Yaskawa INFORM job: X2_38-47,64(2)(90,0).JBI

/JOB
//NAME X2_38-47,64(2)(90,0)
//POS
///NPOS 774,774,774,27,0,0
///TOOL 0
///POSTYPE PULSE
///PULSE
C00000=-10776,-116726,-133110,1428,79202,268
C00001=-117551,-99167,-129064,14869,107235,27560
C00002=-118060,-97833,-124544,14759,105287,27149
C00003=-118255,-97731,-122391,14687,104086,26936
C00004=-118255,-99005,-121658,14606,103015,26804
C00005=-118252,-98719,-121832,14623,103261,26835
C00006=-118753,-92238,-119382,14829,105109,26899
C00007=-118252,-98719,-121832,14623,103261,26835
C00008=-117548,-101379,-128390,14732,105732,27372
C00009=-119930,-99721,-129265,15188,107465,26816
C00010=-120369,-98285,-124713,15062,105542,26424
C00011=-120537,-98252,-122491,14975,104264,26206
C00012=-120537,-99415,-121812,14899,103281,26083
C00013=-120552,-99088,-121997,14922,103557,26112
C00014=-120983,-92542,-119530,15124,105413,26206
C00015=-120552,-99088,-121997,14922,103557,26112
C00016=-119945,-101871,-128593,15052,105999,26622
C00017=-126449,-117484,-130445,19479,74849,30062
C00018=-126433,-122162,-123583,20167,68593,29001
C00019=-126700,-111661,-117040,20113,69946,29141
C00020=-126798,-108107,-114012,20160,69935,29102
C00021=-126799,-108400,-113008,20254,69212,28975
C00022=-126718,-108336,-113627,20168,69582,29070
C00023=-124486,-105728,-112699,19107,69790,29924
C00024=-126718,-108336,-113627,20168,69582,29070
C00025=-121607,-132044,-121280,18982,61321,29585
C00026=-106120,-105771,-112642,10491,66484,36125
C00027=-107709,-101450,-111061,11179,67916,35692
C00028=-106120,-105771,-112642,10491,66484,36125
C00029=-113778,-131562,-126460,14735,63009,32904
C00030=-125989,-135705,-128836,15868,81833,-19678
C00031=-122637,-125595,-122855,15098,82666,-18409
C00032=-121382,-121958,-120533,14807,82865,-17952
C00033=-121382,-122071,-118910,14836,81841,-18076
C00034=-121382,-121958,-120533,14807,82865,-17952
C00035=-106979,-143901,-125029,2861,68009,-11090
C00036=-108002,-136905,-123073,3147,70435,-11396
C00037=-106979,-143901,-125029,2861,68009,-11090
C00038=-130918,-93362,-108301,23503,98063,-21430
C00039=-128613,-93045,-108174,23197,97523,-20724
C00040=-130918,-93362,-108301,23503,98063,-21430
C00041=-136165,-97259,-113946,24281,100844,-22722
C00042=-136175,-89641,-119549,25205,107565,-21267
C00043=-114744,-130738,-127344,-18726,86415,24127
C00044=-118651,-123075,-122041,-18017,86194,22796
C00045=-120132,-120263,-119410,-17742,85711,22351
C00046=-120132,-120365,-118339,-17753,85031,22450
C00047=-120131,-120316,-118616,-17749,85218,22423
C00048=-120610,-114014,-116540,-17635,86988,22001
C00049=-120131,-120316,-118616,-17749,85218,22423
C00050=-120535,-116966,-117470,-17658,86102,22155
C00051=-123144,-118008,-117813,-17156,85246,21372
C00052=-120535,-116966,-117470,-17658,86102,22155
C00053=-115268,-126863,-124750,-18631,86672,23904
C00054=-115290,-123417,-132013,-18678,92595,22992
C00055=-123593,-125758,-130163,6995,115060,-67946
C00056=-111289,-112434,-124190,9231,117016,-63234
C00057=-105837,-112853,-120878,9823,114178,-61462
C00058=-105837,-113368,-119803,9744,113264,-61541
C00059=-105837,-112984,-120626,9804,113958,-61481
C00060=-104314,-115180,-121361,9954,113110,-60999
C00061=-105837,-112984,-120626,9804,113958,-61481
C00062=-140180,-156270,-135194,3647,103600,-74458
C00063=-143876,-158808,-133483,2421,103143,-75779
C00064=-143876,-157752,-132173,2418,102880,-75785
C00065=-143876,-158999,-133717,2421,103190,-75779
C00066=-142833,-166242,-135523,2599,100548,-75469
C00067=-143876,-158999,-133717,2421,103190,-75779
C00068=-138517,-137739,-134524,3768,114393,-73549
C00069=-143641,-117492,-131018,10110,103710,-40081
C00070=-127017,-112123,-129453,9078,98380,-24722
C00071=-128303,-122732,-125182,9622,82824,-11347
C00072=-126354,-112603,-118881,9097,83916,-10616
C00073=-125631,-108986,-116438,8904,84188,-10357
C00074=-125631,-109537,-114964,8919,83013,-10441
C00075=-125631,-108986,-116438,8904,84188,-10357
C00076=-110037,-120252,-118594,-5441,76700,-4050
C00077=-111650,-115152,-116920,-4919,78183,-4659
C00078=-110037,-120252,-118594,-5441,76700,-4050
C00079=-125797,-107165,-114352,8951,83863,-10435
C00080=-123589,-104463,-113383,8361,84418,-9668
C00081=-125797,-107165,-114352,8951,83863,-10435
C00082=-128447,-120300,-122969,9661,82730,-11402
C00083=-128462,-115265,-129707,9620,89375,-10895
C00084=-116938,-126430,-125851,-12631,81878,14685
C00085=-119474,-116309,-119688,-11957,82879,13726
C00086=-120416,-112800,-116898,-11714,82830,13413
C00087=-120416,-113088,-115771,-11732,82005,13491
C00088=-121130,-109897,-115487,-11517,83341,13125
C00089=-121652,-107697,-114715,-11371,83913,12898
C00090=-120385,-110630,-116263,-11708,83544,13356
C00091=-116898,-126708,-125088,-12658,81285,14759
C00092=-116961,-121523,-133241,-12544,88781,13978
C00093=-110477,-156196,-127656,-40514,54336,55405
C00094=-116757,-147091,-123275,-37008,53079,52657
C00095=-119129,-143495,-121504,-35581,52690,51595
C00096=-122199,-143523,-121511,-34086,51426,50520
C00097=-119129,-143495,-121504,-35581,52690,51595
C00098=-121389,-143526,-121523,-34489,51757,50806
C00099=-121378,-138155,-118828,-34021,52680,50458
C00100=-121389,-143526,-121523,-34489,51757,50806
C00101=-121337,-120057,-120260,-30579,61379,47564
C00102=-120272,-114318,-116759,-30898,62447,47698
C00103=-120254,-119054,-117181,-31500,60580,48280
C00104=-120272,-114318,-116759,-30898,62447,47698
C00105=-110477,-159292,-131347,-40206,54861,55162
C00106=-115322,-144881,-127675,-10917,26238,44128
C00107=-131784,-127965,-127002,28991,89678,26741
C00108=-120831,-123140,-121731,27130,85392,29797
C00109=-120549,-120601,-118843,27089,84879,29783
C00110=-120549,-120670,-117777,27109,84260,29640
C00111=-120517,-120686,-117908,27101,84315,29665
C00112=-120983,-114470,-115866,27142,86197,29928
C00113=-120517,-120686,-117908,27101,84315,29665
C00114=-121539,-130455,-126219,27290,84728,29379
C00115=-123491,-138727,-133578,17593,86073,29901
C00116=-123873,-130565,-127363,17655,86508,29830
C00117=-124019,-127789,-124130,17687,86001,29706
C00118=-124019,-127817,-123341,17694,85524,29637
C00119=-124041,-127842,-123499,17696,85609,29642
C00120=-124402,-120732,-121277,17740,87868,29843
C00121=-124041,-127842,-123499,17696,85609,29642
C00122=-123895,-130695,-125894,17671,85585,29689
C00123=-123514,-138829,-132098,17610,85158,29761
C00124=-131669,-108309,-130646,31875,113573,61343
C00125=-139138,-132176,-121475,37127,109735,76690
C00126=-136347,-141301,-121131,36509,104575,76083
C00127=-135137,-144527,-120818,36387,102556,75910
C00128=-135139,-143303,-118803,36292,102059,75739
C00129=-135137,-144527,-120818,36387,102556,75910
C00130=-123222,-117207,-112602,33876,112841,80142
C00131=-123302,-123100,-114500,33386,111310,79603
C00132=-123222,-117207,-112602,33876,112841,80142
C00133=-149473,-167599,-122340,40123,93659,70303
C00134=-145955,-169881,-122827,40768,91382,70949
C00135=-149473,-167599,-122340,40123,93659,70303
C00136=-154660,-158984,-124630,39692,100555,70658
C00137=-145602,-129354,-130944,11561,117970,66438
C00138=-141571,-135796,-129141,-17923,112920,58745
C00139=-145358,-145317,-128855,-18021,107261,58200
C00140=-146973,-148537,-128532,-18134,105137,57926
C00141=-146977,-147425,-126561,-18072,104525,58019
C00142=-146951,-147398,-126788,-18082,104677,58005
C00143=-148016,-155121,-128806,-18044,101844,58047
C00144=-146951,-147398,-126788,-18082,104677,58005
C00145=-147811,-154474,-129578,-18071,102659,57998
C00146=-150760,-151393,-128781,-18698,103033,56852
C00147=-147811,-154474,-129578,-18071,102659,57998
C00148=-142197,-142429,-130522,-17697,110344,58914
C00149=-120703,-123129,-132845,19094,121060,67264
C00150=-120658,-146832,-128060,18624,118943,66884
C00151=-120634,-158899,-128202,17585,113113,65913
C00152=-120623,-163194,-128036,17271,110903,65572
C00153=-120623,-161024,-125795,17237,110651,65534
C00154=-120562,-161261,-126266,17282,110799,65580
C00155=-120543,-169070,-128088,16945,108025,65171
C00156=-120562,-161261,-126266,17282,110799,65580
C00157=-120603,-145779,-126506,18564,118536,66834
C00158=-125859,-133715,-124767,32608,106843,81797
C00159=-122845,-142953,-124347,32149,101432,81430
C00160=-121547,-146160,-123992,32074,99345,81353
C00161=-121546,-144979,-121994,32008,98813,81200
C00162=-109812,-115651,-114700,28773,111647,86169
C00163=-109420,-121743,-116686,28433,109829,85843
C00164=-109812,-115651,-114700,28773,111647,86169
C00165=-136113,-171916,-125823,37236,88758,74782
C00166=-132431,-173177,-126093,37775,86796,75630
C00167=-136113,-171916,-125823,37236,88758,74782
C00168=-141699,-164023,-128432,36630,95711,74814
C00169=-125872,-133752,-131219,33440,110189,40846
C00170=-133109,-126295,-132836,15576,121717,-49477
C00171=-134095,-144484,-127159,11413,120192,-39245
C00172=-134095,-142728,-123587,11251,118920,-39381
C00173=-134108,-141028,-121891,11256,119008,-39376
C00174=-115660,-122947,-115610,-13186,126131,-57848
C00175=-119844,-134491,-118750,-17115,121000,-60623
C00176=-133528,-137451,-116046,-34139,108998,-80448
C00177=-134077,-138654,-116284,-35996,107959,-82962
C00178=-134074,-140235,-119255,-36225,108790,-83252
C00179=-128746,-104991,-133081,-28169,117444,-49732
C00180=-123335,-90933,-122081,-14660,102496,-9308
C00181=-120623,-92535,-112214,-7385,88125,11837
C00182=-120622,-94347,-109953,-7392,85821,11972
C00183=-121706,-96320,-109727,-7087,84579,11689
C00184=-119347,-92925,-108176,-7759,85570,12397
C00185=-120623,-94767,-108750,-7400,84873,12029
C00186=-120184,-98406,-104184,11463,70199,-7234
C00187=-120621,-97250,-102226,16251,67423,-11647
C00188=-120622,-96877,-104163,16104,68755,-11460
C00189=-120643,-108357,-118989,16415,66098,-11840
C00190=-67024,-106779,-124945,-13769,92672,20129
C00191=-67015,-109280,-122780,-13735,90127,20415
C00192=-68524,-114997,-123393,-13374,87393,20218
C00193=-67240,-109374,-121326,-13663,89172,20449
C00194=-67101,-109000,-122679,-13716,90193,20379
C00195=-67110,-106486,-124839,-13750,92741,20094
C00196=-120616,-103713,-129855,-8435,78518,79847
C00197=-120615,-108904,-127553,-8566,74477,80127
C00198=-120827,-110646,-126375,-8530,72852,80171
C00199=-120813,-110572,-126430,-8535,72927,80169
C00200=-120709,-110247,-126307,-8582,73030,80199
C00201=-120779,-110557,-126444,-8550,72945,80181
C00202=-120615,-108909,-127550,-8566,74473,80128
C00203=-118661,-125998,-116417,-35444,53464,49551
C00204=-120918,-122974,-114552,-34038,52889,48644
C00205=-120869,-128815,-114683,-35350,50480,49611
C00206=-120575,-146473,-114035,-40240,44023,53993
C00207=-120599,-119966,-113452,-30276,65744,57931
C00208=-118319,-121507,-115012,-31110,66714,58605
C00209=-113281,-124998,-118777,-32819,69049,60013
C00210=-113467,-117261,-128448,-33027,70743,59318
C00211=-117537,-116112,-134646,-12805,84442,25722
C00212=-120610,-126431,-125414,1040,80197,3464
C00213=-120610,-126707,-122448,1046,78230,3447
C00214=-122238,-127010,-121321,1494,77406,2886
C00215=-120610,-126687,-121221,1049,77486,3441
C00216=-120610,-126294,-121087,1045,77585,3442
C00217=-120610,-126285,-120333,4549,75913,-5215
C00218=-120610,-126340,-121533,4537,76621,-5189
C00219=-125895,-134934,-128716,6057,76967,-6982
C00220=-120648,-124280,-131590,4464,45149,-4941
C00221=-120660,-101129,-132257,5341,102721,-45112
C00222=-120607,-133883,-126281,5735,119700,-79532
C00223=-120606,-133398,-123219,5634,118073,-79618
C00224=-121084,-133632,-122119,5424,117305,-79842
C00225=-121025,-133506,-122086,5447,117346,-79817
C00226=-120605,-133184,-121944,5595,117401,-79652
C00227=-120606,-133121,-120429,13889,116737,-67437
C00228=-120606,-132780,-121444,14001,117514,-67337
C00229=-120606,-133413,-124386,14219,118956,-67146
C00230=-118302,-128282,-130929,25956,92288,-30440
C00231=-120609,-125694,-119256,16594,71477,-14811
C00232=-120609,-125321,-116628,16727,70109,-15005
C00233=-120267,-125069,-115718,16650,69625,-14949
C00234=-120609,-125952,-120025,-8845,76809,6022
C00235=-120609,-125682,-119997,-8842,76927,6012
C00236=-120946,-125172,-117915,-18180,76717,18969
C00237=-120609,-125456,-118894,-18238,77226,19012
C00238=-120610,-125544,-121647,-18141,78796,18775
C00239=-120644,-111765,-129409,-18832,94472,5338
C00240=-120647,-108820,-131188,-26213,120818,-60808
C00241=-120603,-141811,-125437,-24145,112419,-84195
C00242=-120603,-140407,-122244,-23914,111279,-83943
C00243=-120716,-139436,-120851,-23880,110920,-83910
C00244=-120603,-141515,-124307,-1,115345,-75490
C00245=-120603,-141196,-124279,-1,115492,-75490
C00246=-120750,-138616,-117883,30210,107343,-65244
C00247=-120602,-139074,-119094,30337,107734,-65073
C00248=-120603,-140473,-121905,30531,108612,-64825
C00249=-123038,-137969,-128708,31970,112888,-64779
C00250=-147472,-118060,-121113,40576,103304,-81843
C00251=-147472,-118630,-118217,40218,101703,-82475
C00252=-147472,-118727,-117017,40094,101093,-82713
C00253=-147408,-115266,-125424,616,120610,-87255
C00254=-147440,-115512,-125518,608,120541,-87267
C00255=-147454,-115617,-125558,7144,119076,-75809
C00256=-147463,-115686,-125590,12209,115534,-64774
C00257=-147467,-115708,-125608,15036,110623,-54333
C00258=-147465,-115687,-125611,15580,106535,-46817
C00259=-147461,-115654,-125607,15271,104034,-42312
C00260=-147458,-115622,-125603,14500,101619,-37854
C00261=-147455,-115603,-125598,14501,101625,-37852
C00262=-147455,-114670,-126645,14574,102714,-37720
C00263=-147454,-112308,-128585,14752,105047,-37432
C00264=-120607,-127649,-132770,-5702,79300,5510
C00265=-120610,-123519,-126906,-5727,77820,5577
C00266=-120610,-124347,-124400,-5769,75861,5668
C00267=-121328,-123636,-123053,-5535,75349,5445
C00268=-120611,-123827,-123148,-12249,77590,12361
C00269=-120610,-124176,-124804,-8835,80309,9900
C00270=-120610,-124421,-124355,885,77124,6939
C00271=-120609,-123606,-124090,-1533,77411,9469
C00272=-116475,-118028,-122311,-2829,79291,10818
C00273=-112174,-113451,-120859,-4161,80928,12195
C00274=-109550,-110906,-119998,-4966,81848,13023
C00275=-120610,-123835,-125318,-1528,78049,9462
C00276=-120610,-122990,-127374,-1521,79748,9441
C00277=2000,-133752,-131219,0,47993,0
C00278=-10776,-116726,-133110,1428,79202,268
C00279=-117551,-99167,-129064,14869,107235,27560
C00280=-118060,-97833,-124544,14759,105287,27149
C00281=-118255,-97731,-122391,14687,104086,26936
C00282=-118255,-99005,-121658,14606,103015,26804
C00283=-118252,-98719,-121832,14623,103261,26835
C00284=-118753,-92238,-119382,14829,105109,26899
C00285=-118252,-98719,-121832,14623,103261,26835
C00286=-117548,-101379,-128390,14732,105732,27372
C00287=-119930,-99721,-129265,15188,107465,26816
C00288=-120369,-98285,-124713,15062,105542,26424
C00289=-120537,-98252,-122491,14975,104264,26206
C00290=-120537,-99415,-121812,14899,103281,26083
C00291=-120552,-99088,-121997,14922,103557,26112
C00292=-120983,-92542,-119530,15124,105413,26206
C00293=-120552,-99088,-121997,14922,103557,26112
C00294=-119945,-101871,-128593,15052,105999,26622
C00295=-126449,-117484,-130445,19479,74849,30062
C00296=-126433,-122162,-123583,20167,68593,29001
C00297=-126700,-111661,-117040,20113,69946,29141
C00298=-126798,-108107,-114012,20160,69935,29102
C00299=-126799,-108400,-113008,20254,69212,28975
C00300=-126718,-108336,-113627,20168,69582,29070
C00301=-124486,-105728,-112699,19107,69790,29924
C00302=-126718,-108336,-113627,20168,69582,29070
C00303=-121607,-132044,-121280,18982,61321,29585
C00304=-106120,-105771,-112642,10491,66484,36125
C00305=-107709,-101450,-111061,11179,67916,35692
C00306=-106120,-105771,-112642,10491,66484,36125
C00307=-113778,-131562,-126460,14735,63009,32904
C00308=-125989,-135705,-128836,15868,81833,-19678
C00309=-122637,-125595,-122855,15098,82666,-18409
C00310=-121382,-121958,-120533,14807,82865,-17952
C00311=-121382,-122071,-118910,14836,81841,-18076
C00312=-121382,-121958,-120533,14807,82865,-17952
C00313=-106979,-143901,-125029,2861,68009,-11090
C00314=-108002,-136905,-123073,3147,70435,-11396
C00315=-106979,-143901,-125029,2861,68009,-11090
C00316=-130918,-93362,-108301,23503,98063,-21430
C00317=-128613,-93045,-108174,23197,97523,-20724
C00318=-130918,-93362,-108301,23503,98063,-21430
C00319=-136165,-97259,-113946,24281,100844,-22722
C00320=-136175,-89641,-119549,25205,107565,-21267
C00321=-114744,-130738,-127344,-18726,86415,24127
C00322=-118651,-123075,-122041,-18017,86194,22796
C00323=-120132,-120263,-119410,-17742,85711,22351
C00324=-120132,-120365,-118339,-17753,85031,22450
C00325=-120131,-120316,-118616,-17749,85218,22423
C00326=-120610,-114014,-116540,-17635,86988,22001
C00327=-120131,-120316,-118616,-17749,85218,22423
C00328=-120535,-116966,-117470,-17658,86102,22155
C00329=-123144,-118008,-117813,-17156,85246,21372
C00330=-120535,-116966,-117470,-17658,86102,22155
C00331=-115268,-126863,-124750,-18631,86672,23904
C00332=-115290,-123417,-132013,-18678,92595,22992
C00333=-123593,-125758,-130163,6995,115060,-67946
C00334=-111289,-112434,-124190,9231,117016,-63234
C00335=-105837,-112853,-120878,9823,114178,-61462
C00336=-105837,-113368,-119803,9744,113264,-61541
C00337=-105837,-112984,-120626,9804,113958,-61481
C00338=-104314,-115180,-121361,9954,113110,-60999
C00339=-105837,-112984,-120626,9804,113958,-61481
C00340=-140180,-156270,-135194,3647,103600,-74458
C00341=-143876,-158808,-133483,2421,103143,-75779
C00342=-143876,-157752,-132173,2418,102880,-75785
C00343=-143876,-158999,-133717,2421,103190,-75779
C00344=-142833,-166242,-135523,2599,100548,-75469
C00345=-143876,-158999,-133717,2421,103190,-75779
C00346=-138517,-137739,-134524,3768,114393,-73549
C00347=-143641,-117492,-131018,10110,103710,-40081
C00348=-127017,-112123,-129453,9078,98380,-24722
C00349=-128303,-122732,-125182,9622,82824,-11347
C00350=-126354,-112603,-118881,9097,83916,-10616
C00351=-125631,-108986,-116438,8904,84188,-10357
C00352=-125631,-109537,-114964,8919,83013,-10441
C00353=-125631,-108986,-116438,8904,84188,-10357
C00354=-110037,-120252,-118594,-5441,76700,-4050
C00355=-111650,-115152,-116920,-4919,78183,-4659
C00356=-110037,-120252,-118594,-5441,76700,-4050
C00357=-125797,-107165,-114352,8951,83863,-10435
C00358=-123589,-104463,-113383,8361,84418,-9668
C00359=-125797,-107165,-114352,8951,83863,-10435
C00360=-128447,-120300,-122969,9661,82730,-11402
C00361=-128462,-115265,-129707,9620,89375,-10895
C00362=-116938,-126430,-125851,-12631,81878,14685
C00363=-119474,-116309,-119688,-11957,82879,13726
C00364=-120416,-112800,-116898,-11714,82830,13413
C00365=-120416,-113088,-115771,-11732,82005,13491
C00366=-121130,-109897,-115487,-11517,83341,13125
C00367=-121652,-107697,-114715,-11371,83913,12898
C00368=-120385,-110630,-116263,-11708,83544,13356
C00369=-116898,-126708,-125088,-12658,81285,14759
C00370=-116961,-121523,-133241,-12544,88781,13978
C00371=-110477,-156196,-127656,-40514,54336,55405
C00372=-116757,-147091,-123275,-37008,53079,52657
C00373=-119129,-143495,-121504,-35581,52690,51595
C00374=-122199,-143523,-121511,-34086,51426,50520
C00375=-119129,-143495,-121504,-35581,52690,51595
C00376=-121389,-143526,-121523,-34489,51757,50806
C00377=-121378,-138155,-118828,-34021,52680,50458
C00378=-121389,-143526,-121523,-34489,51757,50806
C00379=-121337,-120057,-120260,-30579,61379,47564
C00380=-120272,-114318,-116759,-30898,62447,47698
C00381=-120254,-119054,-117181,-31500,60580,48280
C00382=-120272,-114318,-116759,-30898,62447,47698
C00383=-110477,-159292,-131347,-40206,54861,55162
C00384=-115322,-144881,-127675,-10917,26238,44128
C00385=-131784,-127965,-127002,28991,89678,26741
C00386=-120831,-123140,-121731,27130,85392,29797
C00387=-120549,-120601,-118843,27089,84879,29783
C00388=-120549,-120670,-117777,27109,84260,29640
C00389=-120517,-120686,-117908,27101,84315,29665
C00390=-120983,-114470,-115866,27142,86197,29928
C00391=-120517,-120686,-117908,27101,84315,29665
C00392=-121539,-130455,-126219,27290,84728,29379
C00393=-123491,-138727,-133578,17593,86073,29901
C00394=-123873,-130565,-127363,17655,86508,29830
C00395=-124019,-127789,-124130,17687,86001,29706
C00396=-124019,-127817,-123341,17694,85524,29637
C00397=-124041,-127842,-123499,17696,85609,29642
C00398=-124402,-120732,-121277,17740,87868,29843
C00399=-124041,-127842,-123499,17696,85609,29642
C00400=-123895,-130695,-125894,17671,85585,29689
C00401=-123514,-138829,-132098,17610,85158,29761
C00402=-131669,-108309,-130646,31875,113573,61343
C00403=-139138,-132176,-121475,37127,109735,76690
C00404=-136347,-141301,-121131,36509,104575,76083
C00405=-135137,-144527,-120818,36387,102556,75910
C00406=-135139,-143303,-118803,36292,102059,75739
C00407=-135137,-144527,-120818,36387,102556,75910
C00408=-123222,-117207,-112602,33876,112841,80142
C00409=-123302,-123100,-114500,33386,111310,79603
C00410=-123222,-117207,-112602,33876,112841,80142
C00411=-149473,-167599,-122340,40123,93659,70303
C00412=-145955,-169881,-122827,40768,91382,70949
C00413=-149473,-167599,-122340,40123,93659,70303
C00414=-154660,-158984,-124630,39692,100555,70658
C00415=-145602,-129354,-130944,11561,117970,66438
C00416=-141571,-135796,-129141,-17923,112920,58745
C00417=-145358,-145317,-128855,-18021,107261,58200
C00418=-146973,-148537,-128532,-18134,105137,57926
C00419=-146977,-147425,-126561,-18072,104525,58019
C00420=-146951,-147398,-126788,-18082,104677,58005
C00421=-148016,-155121,-128806,-18044,101844,58047
C00422=-146951,-147398,-126788,-18082,104677,58005
C00423=-147811,-154474,-129578,-18071,102659,57998
C00424=-150760,-151393,-128781,-18698,103033,56852
C00425=-147811,-154474,-129578,-18071,102659,57998
C00426=-142197,-142429,-130522,-17697,110344,58914
C00427=-120703,-123129,-132845,19094,121060,67264
C00428=-120658,-146832,-128060,18624,118943,66884
C00429=-120634,-158899,-128202,17585,113113,65913
C00430=-120623,-163194,-128036,17271,110903,65572
C00431=-120623,-161024,-125795,17237,110651,65534
C00432=-120562,-161261,-126266,17282,110799,65580
C00433=-120543,-169070,-128088,16945,108025,65171
C00434=-120562,-161261,-126266,17282,110799,65580
C00435=-120603,-145779,-126506,18564,118536,66834
C00436=-125859,-133715,-124767,32608,106843,81797
C00437=-122845,-142953,-124347,32149,101432,81430
C00438=-121547,-146160,-123992,32074,99345,81353
C00439=-121546,-144979,-121994,32008,98813,81200
C00440=-109812,-115651,-114700,28773,111647,86169
C00441=-109420,-121743,-116686,28433,109829,85843
C00442=-109812,-115651,-114700,28773,111647,86169
C00443=-136113,-171916,-125823,37236,88758,74782
C00444=-132431,-173177,-126093,37775,86796,75630
C00445=-136113,-171916,-125823,37236,88758,74782
C00446=-141699,-164023,-128432,36630,95711,74814
C00447=-125872,-133752,-131219,33440,110189,40846
C00448=-133109,-126295,-132836,15576,121717,-49477
C00449=-134095,-144484,-127159,11413,120192,-39245
C00450=-134095,-142728,-123587,11251,118920,-39381
C00451=-134108,-141028,-121891,11256,119008,-39376
C00452=-115660,-122947,-115610,-13186,126131,-57848
C00453=-119844,-134491,-118750,-17115,121000,-60623
C00454=-133528,-137451,-116046,-34139,108998,-80448
C00455=-134077,-138654,-116284,-35996,107959,-82962
C00456=-134074,-140235,-119255,-36225,108790,-83252
C00457=-128746,-104991,-133081,-28169,117444,-49732
C00458=-123335,-90933,-122081,-14660,102496,-9308
C00459=-120623,-92535,-112214,-7385,88125,11837
C00460=-120622,-94347,-109953,-7392,85821,11972
C00461=-121706,-96320,-109727,-7087,84579,11689
C00462=-119347,-92925,-108176,-7759,85570,12397
C00463=-120623,-94767,-108750,-7400,84873,12029
C00464=-120184,-98406,-104184,11463,70199,-7234
C00465=-120621,-97250,-102226,16251,67423,-11647
C00466=-120622,-96877,-104163,16104,68755,-11460
C00467=-120643,-108357,-118989,16415,66098,-11840
C00468=-67024,-106779,-124945,-13769,92672,20129
C00469=-67015,-109280,-122780,-13735,90127,20415
C00470=-68524,-114997,-123393,-13374,87393,20218
C00471=-67240,-109374,-121326,-13663,89172,20449
C00472=-67101,-109000,-122679,-13716,90193,20379
C00473=-67110,-106486,-124839,-13750,92741,20094
C00474=-120616,-103713,-129855,-8435,78518,79847
C00475=-120615,-108904,-127553,-8566,74477,80127
C00476=-120827,-110646,-126375,-8530,72852,80171
C00477=-120813,-110572,-126430,-8535,72927,80169
C00478=-120709,-110247,-126307,-8582,73030,80199
C00479=-120779,-110557,-126444,-8550,72945,80181
C00480=-120615,-108909,-127550,-8566,74473,80128
C00481=-118661,-125998,-116417,-35444,53464,49551
C00482=-120918,-122974,-114552,-34038,52889,48644
C00483=-120869,-128815,-114683,-35350,50480,49611
C00484=-120575,-146473,-114035,-40240,44023,53993
C00485=-120599,-119966,-113452,-30276,65744,57931
C00486=-118319,-121507,-115012,-31110,66714,58605
C00487=-113281,-124998,-118777,-32819,69049,60013
C00488=-113467,-117261,-128448,-33027,70743,59318
C00489=-117537,-116112,-134646,-12805,84442,25722
C00490=-120610,-126431,-125414,1040,80197,3464
C00491=-120610,-126707,-122448,1046,78230,3447
C00492=-122238,-127010,-121321,1494,77406,2886
C00493=-120610,-126687,-121221,1049,77486,3441
C00494=-120610,-126294,-121087,1045,77585,3442
C00495=-120610,-126285,-120333,4549,75913,-5215
C00496=-120610,-126340,-121533,4537,76621,-5189
C00497=-125895,-134934,-128716,6057,76967,-6982
C00498=-120648,-124280,-131590,4464,45149,-4941
C00499=-120660,-101129,-132257,5341,102721,-45112
C00500=-120607,-133883,-126281,5735,119700,-79532
C00501=-120606,-133398,-123219,5634,118073,-79618
C00502=-121083,-132569,-121808,5443,117663,-79827
C00503=-120607,-132621,-121847,5608,117630,-79641
C00504=-120606,-132785,-121826,5603,117534,-79644
C00505=-120606,-132451,-120233,13920,116954,-67409
C00506=-120606,-132780,-121444,14001,117514,-67337
C00507=-120606,-133413,-124386,14219,118956,-67146
C00508=-118302,-128282,-130929,25956,92288,-30440
C00509=-120609,-125694,-119256,16594,71477,-14811
C00510=-120609,-125321,-116628,16727,70109,-15005
C00511=-120267,-125069,-115718,16650,69625,-14949
C00512=-120609,-125952,-120025,-8845,76809,6022
C00513=-120609,-125682,-119997,-8842,76927,6012
C00514=-120946,-125172,-117915,-18180,76717,18969
C00515=-120609,-125456,-118894,-18238,77226,19012
C00516=-120610,-125544,-121647,-18141,78796,18775
C00517=-120644,-111765,-129409,-18832,94472,5338
C00518=-120647,-108820,-131188,-26213,120818,-60808
C00519=-120603,-141811,-125437,-24145,112419,-84195
C00520=-120603,-140407,-122244,-23914,111279,-83943
C00521=-120716,-139436,-120851,-23880,110920,-83910
C00522=-120603,-141515,-124307,-1,115345,-75490
C00523=-120603,-141196,-124279,-1,115492,-75490
C00524=-120750,-138616,-117883,30210,107343,-65244
C00525=-120602,-139074,-119094,30337,107734,-65073
C00526=-120603,-140473,-121905,30531,108612,-64825
C00527=-123038,-137969,-128708,31970,112888,-64779
C00528=-147472,-118060,-121113,40576,103304,-81843
C00529=-147472,-118630,-118217,40218,101703,-82475
C00530=-147472,-118727,-117017,40094,101093,-82713
C00531=-147408,-115266,-125424,616,120610,-87255
C00532=-147440,-115512,-125518,608,120541,-87267
C00533=-147454,-115617,-125558,7144,119076,-75809
C00534=-147463,-115686,-125590,12209,115534,-64774
C00535=-147467,-115708,-125608,15036,110623,-54333
C00536=-147465,-115687,-125611,15580,106535,-46817
C00537=-147461,-115654,-125607,15271,104034,-42312
C00538=-147458,-115622,-125603,14500,101619,-37854
C00539=-147455,-115603,-125598,14501,101625,-37852
C00540=-147455,-114670,-126645,14574,102714,-37720
C00541=-147454,-112308,-128585,14752,105047,-37432
C00542=-120607,-127649,-132770,-5702,79300,5510
C00543=-120610,-123519,-126906,-5727,77820,5577
C00544=-120610,-124347,-124400,-5769,75861,5668
C00545=-121328,-123636,-123053,-5535,75349,5445
C00546=-120611,-123827,-123148,-12249,77590,12361
C00547=-120610,-124176,-124804,-8835,80309,9900
C00548=-120610,-124421,-124355,885,77124,6939
C00549=-120609,-123606,-124090,-1533,77411,9469
C00550=-116475,-118028,-122311,-2829,79291,10818
C00551=-112174,-113451,-120859,-4161,80928,12195
C00552=-109550,-110906,-119998,-4966,81848,13023
C00553=-120610,-123835,-125318,-1528,78049,9462
C00554=-120610,-122990,-127374,-1521,79748,9441
C00555=2000,-133752,-131219,0,47993,0
C00556=-63459,-114373,-79771,19626,40886,37257
C00557=-120535,67520,37147,4212,69072,67068
C00558=-120830,69446,43417,4422,66227,66858
C00559=-120946,70374,46117,4513,65052,66770
C00560=-120946,70561,47998,4551,63994,66728
C00561=-120946,70374,46117,4513,65052,66770
C00562=-120262,65088,41656,4214,65044,67021
C00563=-120723,68225,45319,4437,64429,66828
C00564=-120262,65088,41656,4214,65044,67021
C00565=-120141,64198,39022,4125,66199,67107
C00566=-119837,62342,32876,3917,69006,67311
C00567=-133022,42545,9302,483,69993,74705
C00568=-133254,43745,14595,601,67354,74612
C00569=-133346,44332,16823,649,66285,74574
C00570=-133347,44228,18372,654,65278,74568
C00571=-133346,44332,16823,649,66285,74574
C00572=-132762,39917,13904,373,65809,74781
C00573=-133123,42775,16905,546,65433,74650
C00574=-132762,39917,13904,373,65809,74781
C00575=-132666,39314,11672,325,66873,74819
C00576=-132425,38068,6360,208,69500,74909
C00577=-155117,5532,-38436,2147,90846,73739
C00578=-181330,90113,53999,1695,94832,75162
C00579=-181479,87228,54387,1703,93114,75089
C00580=-181540,86155,54651,1706,92402,75059
C00581=-181542,86152,56307,1705,91382,75044
C00582=-181540,86155,54651,1706,92402,75059
C00583=-180656,94851,65604,1626,90111,75325
C00584=-181131,94253,66558,1666,89229,75153
C00585=-181349,89885,61022,1686,90394,75096
C00586=-181131,94253,66558,1666,89229,75153
C00587=-181073,95243,66217,1662,89945,75182
C00588=-180930,97948,65680,1651,91663,75253
C00589=-185436,101694,69046,-5553,88631,72150
C00590=-185900,99624,70331,-5496,86754,72076
C00591=-186087,98901,70984,-5475,85971,72047
C00592=-186087,99023,71813,-5476,85523,72066
C00593=-186087,98901,70984,-5475,85971,72047
C00594=-185708,102060,75107,-5528,85087,72214
C00595=-185637,106217,81264,-5546,83447,72310
C00596=-185813,101011,74470,-5516,84934,72189
C00597=-185596,102468,75930,-5543,84801,72264
C00598=-185712,103515,76702,-5528,84853,72223
C00599=-185252,105372,75160,-5578,86780,72294
C00600=-160848,14099,-19058,-268,71131,81958
C00601=-166181,22945,-3449,-1246,81387,-4932
C00602=-165629,27427,7007,-1415,77267,-4702
C00603=-165325,28785,10065,-1509,76088,-4584
C00604=-165325,28859,11250,-1513,75397,-4577
C00605=-165325,28785,10065,-1509,76088,-4584
C00606=-165316,31705,12964,-1515,75805,-4576
C00607=-165325,28785,10065,-1509,76088,-4584
C00608=-158615,35277,16566,-12881,79402,10247
C00609=-158695,35491,17753,-12887,78784,10285
C00610=-159268,36430,18712,-12762,78589,10105
C00611=-158695,35389,16453,-12860,79513,10210
C00612=-158695,35595,7262,-12723,85139,9628
C00613=-159201,23460,163,-1108,64126,82575
C00614=-159224,25290,5934,-1122,61515,82592
C00615=-159868,27923,10103,-801,60293,82359
C00616=-159868,27994,11092,-805,59722,82362
C00617=-159702,23782,6087,-883,60640,82418
C00618=-159324,22038,5481,-1084,60120,82567
C00619=-159393,26328,9606,-1054,59786,82544
C00620=-159613,24178,6270,-930,60732,82451
C00621=-159229,18801,-2529,-1101,63389,82571
C00622=-183717,54594,32393,11335,61848,73349
C00623=-183547,57223,39351,11572,58949,73113
C00624=-183480,58440,42335,11685,57752,73010
C00625=-183483,58871,44494,11828,56667,72889
C00626=-183480,58440,42335,11685,57752,73010
C00627=-183942,52495,37403,11920,57800,72829
C00628=-183665,55840,41125,11854,57199,72874
C00629=-183942,52495,37403,11920,57800,72829
C00630=-184013,51323,34501,11809,58970,72930
C00631=-184190,48769,27698,11575,61813,73164
C00632=-194866,69356,39319,16134,66946,69768
C00633=-193573,77344,52867,16088,62620,69643
C00634=-193573,77518,54262,16198,61881,69535
C00635=-193573,77677,55340,16285,61320,69453
C00636=-193573,77577,54676,16232,61664,69504
C00637=-194136,69418,44929,16234,63513,69555
C00638=-194228,70015,46296,16348,63023,69447
C00639=-193714,74954,52179,16268,61881,69478
C00640=-194171,69155,43983,16191,63957,69605
C00641=-195158,66932,37846,16301,66678,69622
C00642=-181592,-32488,-72920,9217,81357,75741
C00643=-150216,-104680,-71296,-7403,42753,75254
C00644=-146927,-106152,-71782,-9593,42642,76873
C00645=-147684,-69879,-51768,-13743,41767,65179
C00646=-160676,17315,-11357,-3352,97353,79993
C00647=-160891,14623,-4117,-3294,91515,80076
C00648=-160978,13901,-3178,-3284,90564,80072
C00649=-160978,13971,-1710,-3282,89697,80095
C00650=-160978,13901,-3178,-3284,90564,80072
C00651=-160255,23408,5198,-3348,90324,80321
C00652=-160499,21544,5437,-3325,89208,80271
C00653=-160501,19595,3599,-3325,89335,80267
C00654=-160244,20737,3724,-3349,89854,80340
C00655=-160609,22303,808,-3324,92440,80146
C00656=-146158,-25817,-42599,-18441,59324,81079
C00657=-149286,-19659,-34519,-16945,56935,80217
C00658=-149286,-19679,-33192,-17101,56143,80346
C00659=-149286,-19666,-31921,-17254,55400,80472
C00660=-149283,-19680,-33312,-17071,56218,80336
C00661=-148502,-26328,-38062,-17636,55910,80711
C00662=-148502,-26286,-36495,-17832,55009,80867
C00663=-149157,-21917,-33398,-17365,55193,80560
C00664=-149857,-25642,-38896,-16657,56458,80060
C00665=-145616,-30275,-43889,-19038,58025,81528
C00666=-147684,-69879,-51768,-13743,41767,65179
C00667=-146927,-106152,-71782,-9593,42642,76873
C00668=-150216,-104680,-71296,-7403,42753,75254
C00669=-181592,-37651,-66165,9425,74633,75233
C00670=-161871,17303,-4712,10555,76262,79929
C00671=-161452,17546,-388,10536,73713,79854
C00672=-164352,5532,-4911,18132,62198,77732
C00673=-162815,5376,-4950,17454,61813,78279
C00674=-160145,17568,-217,10119,73455,80292
C00675=-160561,17295,-4569,10141,76006,80359
C00676=-160561,17295,-4569,10141,77854,24225
C00677=-154925,3428,-11232,-4624,70900,30462
C00678=-155821,5540,-7163,-4340,69436,30196
C00679=-157012,4626,-7218,-1589,68724,27505
C00680=-155631,5235,-4373,-2115,67316,28026
C00681=-155501,1121,-9941,-2144,68631,28049
C00682=-164062,1653,-9261,9806,70969,1365
C00683=-163111,13453,569,7852,75819,2004
C00684=-169111,38169,24298,20475,87264,-21600
C00685=-171145,34811,19304,20623,89038,-22029
C00686=-170232,24106,-2783,18479,91787,-14288
C00687=-160304,11530,-9767,5228,51358,81447
C00688=-160077,14832,-4280,5183,49670,81455
C00689=-160516,13652,-395,8281,43180,80940
C00690=-159075,15987,128,5765,45857,81735
C00691=-164330,15419,2317,23639,44338,76758
C00692=-163385,18960,-1174,18743,50959,78553
C00693=-165374,13239,-6613,20923,51920,77727
C00694=-161014,13295,-8090,-6406,49355,82824
C00695=-161267,16828,-2191,-6383,47532,82835
C00696=-161514,15510,839,-4919,41379,83326
C00697=-163506,13140,558,-1967,37945,82559
C00698=-158654,12998,2510,-21078,36813,89125
C00699=-156013,15323,-3292,-22041,49335,86873
C00700=-155829,15379,-4520,-22688,50226,86879
C00701=-196408,57492,27109,18880,55161,68375
C00702=-196116,61126,34099,19257,52786,68047
C00703=-196681,60945,37268,23427,49055,67256
C00704=-198137,64293,40871,24244,49217,66577
C00705=-198035,64746,39034,20821,52142,67068
C00706=-198350,60950,31019,20265,55020,67530
C00707=-186747,89870,54733,-990,89142,72486
C00708=-186403,90906,60090,-1045,86383,72625
C00709=-181702,120366,100649,-11275,85103,73801
C00710=-183469,126371,108859,-11233,82931,73387
C00711=-188139,94217,64278,-773,85485,72048
C00712=-188503,92942,58606,-716,88318,71911
C00713=-158356,2052,-43381,6178,92005,68050
C00714=-121453,57439,26725,6551,67570,68970
C00715=-121610,59341,32873,6761,64794,68755
C00716=-121469,44825,24088,7614,53384,68067
C00717=-119406,47984,28011,6377,51946,68833
C00718=-119643,63560,37702,5874,63844,69428
C00719=-119474,61501,31338,5667,66676,69631
C00720=-119468,73784,45718,-1688,68030,70001
C00721=-119896,75838,52185,-1543,65099,69887
C00722=-119734,60370,40471,-1882,55599,70088
C00723=-120784,60524,39839,-1249,57371,69644
C00724=-121139,72676,48393,-1011,65788,69424
C00725=-120714,70771,42130,-1166,68668,69550
C00726=-130022,48445,16791,-5635,70294,75741
C00727=-130464,49596,22041,-5533,67637,75710
C00728=-130594,37241,15185,-4965,57340,76243
C00729=-134757,36577,12787,-2863,61070,74469
C00730=-134997,44020,16033,-3483,68218,74080
C00731=-134574,42926,10871,-3614,70846,74149
C00732=-144116,-100954,-108623,608,70277,70877
C00733=-125234,-105855,-90971,-8573,57832,78294
C00734=-134723,-30987,-43000,-16193,82094,-73445
C00735=-147286,-18641,-32771,2207,85620,-76456
C00736=-145987,-10544,-25760,-132,91452,-76157
C00737=-145688,-12541,-27327,264,90178,-76022
C00738=-147179,-23652,-36397,2189,85274,-76425
C00739=-147575,-22440,-39612,2256,87884,-76511
C00740=-160185,17986,-3976,-6942,87400,-80225
C00741=-160429,16792,-1004,-6911,84954,-80173
C00742=-159753,19362,2506,-7031,84177,-79901
C00743=-161023,19371,2516,-6819,84070,-80326
C00744=-161231,16782,-1016,-6776,84888,-80439
C00745=-160981,17969,-3994,-6807,87335,-80488
C00746=-162074,-26616,-42506,-1763,64705,-79693
C00747=-162070,-24854,-37261,-1799,62384,-79656
C00748=-162385,-21834,-34052,-1646,61952,-79768
C00749=-160369,-21963,-34144,-2676,61996,-79016
C00750=-159769,-24818,-37192,-4027,62449,-78761
C00751=-159682,-26579,-42435,-3993,64769,-78811
C00752=-159749,-26590,-42466,-830,64636,-81339
C00753=-159773,-24828,-37221,-834,62313,-81331
C00754=-159460,-21788,-33850,-1000,61804,-81209
C00755=-160671,-21843,-33924,-379,61812,-81664
C00756=-162116,-24842,-37231,1419,62318,-82243
C00757=-162183,-26603,-42475,1425,64641,-82238
C00758=-125234,-105855,-90971,-8573,57832,78294
C00759=-144116,-100954,-108623,608,70277,70877
C00760=-180054,17730,-13564,7282,57092,75133
C00761=-184405,44193,24876,11651,47654,72434
C00762=-186268,39946,27192,20044,40162,70477
C00763=-189224,45695,31842,20419,42291,69339
C00764=-188153,48497,30967,14785,46766,70568
C00765=-188342,44346,22853,14289,49572,70918
C00766=-179348,87345,51596,-2140,89915,74922
C00767=-179631,85372,53193,-2095,87912,74861
C00768=-176610,100170,73501,-7799,88743,75470
C00769=-180322,105518,80466,-7431,86799,74328
C00770=-183307,90153,59154,-1526,86619,73655
C00771=-183010,91971,57396,-1572,88641,73729
C00772=-153116,42547,-17943,-6513,110885,24646
C00773=-10907,-117335,-90652,-18762,63715,-59495
BC00000=165820,667836,1075229
BC00001=398174,1010261,1075175
BC00002=398174,1010261,1075175
BC00003=398174,1010261,1075175
BC00004=398174,1010261,1075175
BC00005=398174,1010261,1075175
BC00006=398174,1010261,1075175
BC00007=398174,1010261,1075175
BC00008=398174,1010261,1075175
BC00009=355157,1002325,1075175
BC00010=355157,1002325,1075175
BC00011=355157,1002325,1075175
BC00012=355157,1002325,1075175
BC00013=355157,1002325,1075175
BC00014=355157,1002325,1075175
BC00015=355157,1002325,1075175
BC00016=355157,1002325,1075175
BC00017=253987,909376,1075175
BC00018=253987,909376,1075175
BC00019=253987,909376,1075175
BC00020=253987,909376,1075175
BC00021=253987,909376,1075175
BC00022=253987,909376,1075175
BC00023=253987,909376,1075175
BC00024=253987,909376,1075175
BC00025=253987,909376,1075175
BC00026=253987,909376,1075175
BC00027=253987,909376,1075175
BC00028=253987,909376,1075175
BC00029=253987,909376,1075175
BC00030=147037,948855,1075175
BC00031=147037,948855,1075175
BC00032=147037,948855,1075175
BC00033=147037,948855,1075175
BC00034=147037,948855,1075175
BC00035=147037,948855,1075175
BC00036=147037,948855,1075175
BC00037=147037,948855,1075175
BC00038=147037,948855,1075175
BC00039=147037,948855,1075175
BC00040=147037,948855,1075175
BC00041=147037,948855,1075175
BC00042=147037,948855,1075175
BC00043=175618,946621,1075175
BC00044=175618,946621,1075175
BC00045=175618,946621,1075175
BC00046=175618,946621,1075175
BC00047=175618,946621,1075175
BC00048=175618,946621,1075175
BC00049=175618,946621,1075175
BC00050=175618,946621,1075175
BC00051=175618,946621,1075175
BC00052=175618,946621,1075175
BC00053=175618,946621,1075175
BC00054=175618,946621,1075175
BC00055=144312,974949,1075175
BC00056=144312,974949,1075175
BC00057=144312,974949,1075175
BC00058=144312,974949,1075175
BC00059=144312,974949,1075175
BC00060=144312,974949,1075175
BC00061=144312,974949,1075175
BC00062=144312,974949,1075175
BC00063=144312,974949,1075175
BC00064=144312,974949,1075175
BC00065=144312,974949,1075175
BC00066=144312,974949,1075175
BC00067=144312,974949,1075175
BC00068=144312,974949,1075175
BC00069=159928,928652,1075175
BC00070=164440,875523,1075175
BC00071=171034,862645,1075175
BC00072=171034,862645,1075175
BC00073=171034,862645,1075175
BC00074=171034,862645,1075175
BC00075=171034,862645,1075175
BC00076=171034,862645,1075175
BC00077=171034,862645,1075175
BC00078=171034,862645,1075175
BC00079=171034,862645,1075175
BC00080=171034,862645,1075175
BC00081=171034,862645,1075175
BC00082=171034,862645,1075175
BC00083=171034,862645,1075175
BC00084=164738,841983,1075175
BC00085=164738,841983,1075175
BC00086=164738,841983,1075175
BC00087=164738,841983,1075175
BC00088=164738,841983,1075175
BC00089=164738,841983,1075175
BC00090=164738,841983,1075175
BC00091=164738,841983,1075175
BC00092=164738,841983,1075175
BC00093=143339,934688,1075175
BC00094=143339,934688,1075175
BC00095=143339,934688,1075175
BC00096=143339,934688,1075175
BC00097=143339,934688,1075175
BC00098=143339,934688,1075175
BC00099=143339,934688,1075175
BC00100=143339,934688,1075175
BC00101=143339,934688,1075175
BC00102=143339,934688,1075175
BC00103=143339,934688,1075175
BC00104=143339,934688,1075175
BC00105=143339,934688,1075175
BC00106=95192,864025,1075175
BC00107=33067,951094,1075175
BC00108=33067,951094,1075175
BC00109=33067,951094,1075175
BC00110=33067,951094,1075175
BC00111=33067,951094,1075175
BC00112=33067,951094,1075175
BC00113=33067,951094,1075175
BC00114=33067,951094,1075175
BC00115=15,945322,1075175
BC00116=15,945322,1075175
BC00117=15,945322,1075175
BC00118=15,945322,1075175
BC00119=15,945322,1075175
BC00120=15,945322,1075175
BC00121=15,945322,1075175
BC00122=15,945322,1075175
BC00123=15,945322,1075175
BC00124=16460,857819,1075175
BC00125=28300,807028,1075175
BC00126=28300,807028,1075175
BC00127=28300,807028,1075175
BC00128=28300,807028,1075175
BC00129=28300,807028,1075175
BC00130=28300,807028,1075175
BC00131=28300,807028,1075175
BC00132=28300,807028,1075175
BC00133=28300,807028,1075175
BC00134=28300,807028,1075175
BC00135=28300,807028,1075175
BC00136=28300,807028,1075175
BC00137=49949,826856,1075175
BC00138=70323,828866,1075175
BC00139=70323,828866,1075175
BC00140=70323,828866,1075175
BC00141=70323,828866,1075175
BC00142=70323,828866,1075175
BC00143=70323,828866,1075175
BC00144=70323,828866,1075175
BC00145=70323,828866,1075175
BC00146=70323,828866,1075175
BC00147=70323,828866,1075175
BC00148=70323,828866,1075175
BC00149=113400,816475,1075175
BC00150=113400,846295,1075175
BC00151=113400,846295,1075175
BC00152=113400,846295,1075175
BC00153=113400,846295,1075175
BC00154=113400,846295,1075175
BC00155=113400,846295,1075175
BC00156=113400,846295,1075175
BC00157=113400,846295,1075175
BC00158=126179,809480,1075175
BC00159=126179,809480,1075175
BC00160=126179,809480,1075175
BC00161=126179,809480,1075175
BC00162=126179,809480,1075175
BC00163=126179,809480,1075175
BC00164=126179,809480,1075175
BC00165=126179,809480,1075175
BC00166=126179,809480,1075175
BC00167=126179,809480,1075175
BC00168=126179,809480,1075175
BC00169=126179,809480,1075175
BC00170=153260,992688,1075175
BC00171=154894,1008954,1075175
BC00172=159567,1006428,1075175
BC00173=161040,1005633,1075171
BC00174=188180,1004944,1075172
BC00175=159398,988729,1075171
BC00176=196171,985949,1075168
BC00177=201136,987895,1075175
BC00178=203670,993516,1075175
BC00179=184106,924906,1075175
BC00180=164145,855826,1075175
BC00181=154136,821185,1075175
BC00182=151914,826190,1075175
BC00183=151025,828192,1075175
BC00184=151025,828192,1075175
BC00185=197574,854331,1075175
BC00186=160004,840173,1075175
BC00187=151157,834851,1075175
BC00188=148293,828805,1075175
BC00189=148293,828805,1075175
BC00190=312275,994515,1075175
BC00191=311979,999858,1075175
BC00192=311860,1001996,1075175
BC00193=362733,1010828,1075164
BC00194=362852,1008691,1075175
BC00195=363148,1003347,1075175
BC00196=102795,934804,1075175
BC00197=101452,936777,1075175
BC00198=100915,937567,1075175
BC00199=100906,939899,1075175
BC00200=100898,942175,1075175
BC00201=100889,944507,1075175
BC00202=101426,943718,1075175
BC00203=141515,928256,1075175
BC00204=141515,928256,1075175
BC00205=141515,928256,1075175
BC00206=141515,928257,1075172
BC00207=141515,928256,1075175
BC00208=141515,928256,1075175
BC00209=141515,928256,1075175
BC00210=141515,916104,1075175
BC00211=68127,920356,1075175
BC00212=16830,923328,1075175
BC00213=16562,928525,1075175
BC00214=16455,930603,1075175
BC00215=16455,930603,1075175
BC00216=71893,940191,1075175
BC00217=67464,939156,1075175
BC00218=67022,937046,1075175
BC00219=65915,931769,1075175
BC00220=65915,901978,1075175
BC00221=98323,852136,1075175
BC00222=125079,831224,1075175
BC00223=125794,825809,1075175
BC00224=126079,823643,1075174
BC00225=126677,823645,1075174
BC00226=170108,823795,1075173
BC00227=157966,823650,1075175
BC00228=156869,825691,1075175
BC00229=154126,830791,1075175
BC00230=114692,901690,1075175
BC00231=143002,931232,1075175
BC00232=146315,936443,1075175
BC00233=147641,938527,1075175
BC00234=194941,944470,1075175
BC00235=156841,937856,1075175
BC00236=172703,940853,1075175
BC00237=174292,939117,1075175
BC00238=178267,934778,1075175
BC00239=164918,911333,1075175
BC00240=91107,849480,1075175
BC00241=59698,829503,1075175
BC00242=57257,824323,1075175
BC00243=56280,822250,1075175
BC00244=29836,827677,1075175
BC00245=76754,827839,1075175
BC00246=27687,817329,1075175
BC00247=25853,819104,1075175
BC00248=21269,823543,1075175
BC00249=34689,834409,1075171
BC00250=267738,1017378,1075175
BC00251=272730,1015553,1075175
BC00252=274727,1014823,1075175
BC00253=328708,1053146,1075175
BC00254=294162,1033751,1075175
BC00255=279435,1024890,1075175
BC00256=269339,1011255,1075175
BC00257=265430,994958,1075175
BC00258=267336,981721,1075175
BC00259=271332,972471,1075175
BC00260=275026,965943,1075175
BC00261=277522,963553,1075175
BC00262=275862,962700,1075175
BC00263=272541,960996,1075175
BC00264=271715,892373,1073460
BC00265=294826,916334,1075175
BC00266=293545,921932,1075175
BC00267=293032,924172,1075175
BC00268=307043,929007,1075175
BC00269=302586,932369,1075175
BC00270=285695,927618,1075175
BC00271=319756,944028,1075175
BC00272=321000,944625,1075175
BC00273=321000,944625,1075175
BC00274=321000,944625,1075175
BC00275=325770,944528,1075175
BC00276=326754,940227,1075175
BC00277=126179,666204,1075175
BC00278=165820,667836,1075229
BC00279=398174,1010261,1075175
BC00280=398174,1010261,1075175
BC00281=398174,1010261,1075175
BC00282=398174,1010261,1075175
BC00283=398174,1010261,1075175
BC00284=398174,1010261,1075175
BC00285=398174,1010261,1075175
BC00286=398174,1010261,1075175
BC00287=355157,1002325,1075175
BC00288=355157,1002325,1075175
BC00289=355157,1002325,1075175
BC00290=355157,1002325,1075175
BC00291=355157,1002325,1075175
BC00292=355157,1002325,1075175
BC00293=355157,1002325,1075175
BC00294=355157,1002325,1075175
BC00295=253987,909376,1075175
BC00296=253987,909376,1075175
BC00297=253987,909376,1075175
BC00298=253987,909376,1075175
BC00299=253987,909376,1075175
BC00300=253987,909376,1075175
BC00301=253987,909376,1075175
BC00302=253987,909376,1075175
BC00303=253987,909376,1075175
BC00304=253987,909376,1075175
BC00305=253987,909376,1075175
BC00306=253987,909376,1075175
BC00307=253987,909376,1075175
BC00308=147037,948855,1075175
BC00309=147037,948855,1075175
BC00310=147037,948855,1075175
BC00311=147037,948855,1075175
BC00312=147037,948855,1075175
BC00313=147037,948855,1075175
BC00314=147037,948855,1075175
BC00315=147037,948855,1075175
BC00316=147037,948855,1075175
BC00317=147037,948855,1075175
BC00318=147037,948855,1075175
BC00319=147037,948855,1075175
BC00320=147037,948855,1075175
BC00321=175618,946621,1075175
BC00322=175618,946621,1075175
BC00323=175618,946621,1075175
BC00324=175618,946621,1075175
BC00325=175618,946621,1075175
BC00326=175618,946621,1075175
BC00327=175618,946621,1075175
BC00328=175618,946621,1075175
BC00329=175618,946621,1075175
BC00330=175618,946621,1075175
BC00331=175618,946621,1075175
BC00332=175618,946621,1075175
BC00333=144312,974949,1075175
BC00334=144312,974949,1075175
BC00335=144312,974949,1075175
BC00336=144312,974949,1075175
BC00337=144312,974949,1075175
BC00338=144312,974949,1075175
BC00339=144312,974949,1075175
BC00340=144312,974949,1075175
BC00341=144312,974949,1075175
BC00342=144312,974949,1075175
BC00343=144312,974949,1075175
BC00344=144312,974949,1075175
BC00345=144312,974949,1075175
BC00346=144312,974949,1075175
BC00347=159928,928652,1075175
BC00348=164440,875523,1075175
BC00349=171034,862645,1075175
BC00350=171034,862645,1075175
BC00351=171034,862645,1075175
BC00352=171034,862645,1075175
BC00353=171034,862645,1075175
BC00354=171034,862645,1075175
BC00355=171034,862645,1075175
BC00356=171034,862645,1075175
BC00357=171034,862645,1075175
BC00358=171034,862645,1075175
BC00359=171034,862645,1075175
BC00360=171034,862645,1075175
BC00361=171034,862645,1075175
BC00362=164738,841983,1075175
BC00363=164738,841983,1075175
BC00364=164738,841983,1075175
BC00365=164738,841983,1075175
BC00366=164738,841983,1075175
BC00367=164738,841983,1075175
BC00368=164738,841983,1075175
BC00369=164738,841983,1075175
BC00370=164738,841983,1075175
BC00371=143339,934688,1075175
BC00372=143339,934688,1075175
BC00373=143339,934688,1075175
BC00374=143339,934688,1075175
BC00375=143339,934688,1075175
BC00376=143339,934688,1075175
BC00377=143339,934688,1075175
BC00378=143339,934688,1075175
BC00379=143339,934688,1075175
BC00380=143339,934688,1075175
BC00381=143339,934688,1075175
BC00382=143339,934688,1075175
BC00383=143339,934688,1075175
BC00384=95192,864025,1075175
BC00385=33067,951094,1075175
BC00386=33067,951094,1075175
BC00387=33067,951094,1075175
BC00388=33067,951094,1075175
BC00389=33067,951094,1075175
BC00390=33067,951094,1075175
BC00391=33067,951094,1075175
BC00392=33067,951094,1075175
BC00393=15,945322,1075175
BC00394=15,945322,1075175
BC00395=15,945322,1075175
BC00396=15,945322,1075175
BC00397=15,945322,1075175
BC00398=15,945322,1075175
BC00399=15,945322,1075175
BC00400=15,945322,1075175
BC00401=15,945322,1075175
BC00402=16460,857819,1075175
BC00403=28300,807028,1075175
BC00404=28300,807028,1075175
BC00405=28300,807028,1075175
BC00406=28300,807028,1075175
BC00407=28300,807028,1075175
BC00408=28300,807028,1075175
BC00409=28300,807028,1075175
BC00410=28300,807028,1075175
BC00411=28300,807028,1075175
BC00412=28300,807028,1075175
BC00413=28300,807028,1075175
BC00414=28300,807028,1075175
BC00415=49949,826856,1075175
BC00416=70323,828866,1075175
BC00417=70323,828866,1075175
BC00418=70323,828866,1075175
BC00419=70323,828866,1075175
BC00420=70323,828866,1075175
BC00421=70323,828866,1075175
BC00422=70323,828866,1075175
BC00423=70323,828866,1075175
BC00424=70323,828866,1075175
BC00425=70323,828866,1075175
BC00426=70323,828866,1075175
BC00427=113400,816475,1075175
BC00428=113400,846295,1075175
BC00429=113400,846295,1075175
BC00430=113400,846295,1075175
BC00431=113400,846295,1075175
BC00432=113400,846295,1075175
BC00433=113400,846295,1075175
BC00434=113400,846295,1075175
BC00435=113400,846295,1075175
BC00436=126179,809480,1075175
BC00437=126179,809480,1075175
BC00438=126179,809480,1075175
BC00439=126179,809480,1075175
BC00440=126179,809480,1075175
BC00441=126179,809480,1075175
BC00442=126179,809480,1075175
BC00443=126179,809480,1075175
BC00444=126179,809480,1075175
BC00445=126179,809480,1075175
BC00446=126179,809480,1075175
BC00447=126179,809480,1075175
BC00448=153260,992688,1075175
BC00449=154894,1008954,1075175
BC00450=159567,1006428,1075175
BC00451=161040,1005633,1075171
BC00452=188180,1004944,1075172
BC00453=159398,988729,1075171
BC00454=196171,985949,1075168
BC00455=201136,987895,1075175
BC00456=203670,993516,1075175
BC00457=184106,924906,1075175
BC00458=164145,855826,1075175
BC00459=154136,821185,1075175
BC00460=151914,826190,1075175
BC00461=151025,828192,1075175
BC00462=151025,828192,1075175
BC00463=197574,854331,1075175
BC00464=160004,840173,1075175
BC00465=151157,834851,1075175
BC00466=148293,828805,1075175
BC00467=148293,828805,1075175
BC00468=312275,994515,1075175
BC00469=311979,999858,1075175
BC00470=311860,1001996,1075175
BC00471=362733,1010828,1075164
BC00472=362852,1008691,1075175
BC00473=363148,1003347,1075175
BC00474=102795,934804,1075175
BC00475=101452,936777,1075175
BC00476=100915,937567,1075175
BC00477=100906,939899,1075175
BC00478=100898,942175,1075175
BC00479=100889,944507,1075175
BC00480=101426,943718,1075175
BC00481=141515,928256,1075175
BC00482=141515,928256,1075175
BC00483=141515,928256,1075175
BC00484=141515,928257,1075172
BC00485=141515,928256,1075175
BC00486=141515,928256,1075175
BC00487=141515,928256,1075175
BC00488=141515,916104,1075175
BC00489=68127,920356,1075175
BC00490=16830,923328,1075175
BC00491=16562,928525,1075175
BC00492=16455,930603,1075175
BC00493=16455,930603,1075175
BC00494=71893,940191,1075175
BC00495=67464,939156,1075175
BC00496=67022,937046,1075175
BC00497=65915,931769,1075175
BC00498=65915,901978,1075175
BC00499=98323,852136,1075175
BC00500=125079,831224,1075175
BC00501=125794,825809,1075175
BC00502=126079,823643,1075175
BC00503=130858,823659,1075175
BC00504=170108,823795,1075173
BC00505=157966,823650,1075175
BC00506=156869,825691,1075175
BC00507=154126,830791,1075175
BC00508=114692,901690,1075175
BC00509=143002,931232,1075175
BC00510=146315,936443,1075175
BC00511=147641,938527,1075175
BC00512=194941,944470,1075175
BC00513=156841,937856,1075175
BC00514=172703,940853,1075175
BC00515=174292,939117,1075175
BC00516=178267,934778,1075175
BC00517=164918,911333,1075175
BC00518=91107,849480,1075175
BC00519=59698,829503,1075175
BC00520=57257,824323,1075175
BC00521=56280,822250,1075175
BC00522=29836,827677,1075175
BC00523=76754,827839,1075175
BC00524=27687,817329,1075175
BC00525=25853,819104,1075175
BC00526=21269,823543,1075175
BC00527=34689,834409,1075171
BC00528=267738,1017378,1075175
BC00529=272730,1015553,1075175
BC00530=274727,1014823,1075175
BC00531=328708,1053146,1075175
BC00532=294162,1033751,1075175
BC00533=279435,1024890,1075175
BC00534=269339,1011255,1075175
BC00535=265430,994958,1075175
BC00536=267336,981721,1075175
BC00537=271332,972471,1075175
BC00538=275026,965943,1075175
BC00539=277522,963553,1075175
BC00540=275862,962700,1075175
BC00541=272541,960996,1075175
BC00542=271715,892373,1073460
BC00543=294826,916334,1075175
BC00544=293545,921932,1075175
BC00545=293032,924172,1075175
BC00546=307043,929007,1075175
BC00547=302586,932369,1075175
BC00548=285695,927618,1075175
BC00549=319756,944028,1075175
BC00550=321000,944625,1075175
BC00551=321000,944625,1075175
BC00552=321000,944625,1075175
BC00553=325770,944528,1075175
BC00554=326754,940227,1075175
BC00555=126179,666204,1075175
BC00556=216726,717474,641306
BC00557=301368,789553,152612
BC00558=301368,789553,152612
BC00559=301368,789553,152612
BC00560=301368,789553,152612
BC00561=301368,789553,152612
BC00562=301368,789553,152612
BC00563=301368,789553,152612
BC00564=301368,789553,152612
BC00565=301368,789553,152612
BC00566=301368,789553,152612
BC00567=314485,789553,143111
BC00568=314485,789553,143111
BC00569=314485,789553,143111
BC00570=314485,789553,143111
BC00571=314485,789553,143111
BC00572=314485,789553,143111
BC00573=314485,789553,143111
BC00574=314485,789553,143111
BC00575=314485,789553,143111
BC00576=314485,789553,143111
BC00577=331615,789553,138281
BC00578=360333,789553,130184
BC00579=360333,789553,130184
BC00580=360333,789553,130184
BC00581=360333,789553,130184
BC00582=360333,789553,130184
BC00583=360333,789553,130184
BC00584=360333,789553,130184
BC00585=360333,789553,130184
BC00586=360333,789553,130184
BC00587=360333,789553,130184
BC00588=360333,789553,130184
BC00589=360105,789553,124885
BC00590=360105,789553,124885
BC00591=360105,789553,124885
BC00592=360105,789553,124885
BC00593=360105,789553,124885
BC00594=360105,789553,124885
BC00595=360105,789553,124885
BC00596=360105,789553,124885
BC00597=360105,789553,124885
BC00598=360105,789553,124885
BC00599=360105,789553,124885
BC00600=345851,783755,200789
BC00601=345851,783755,200789
BC00602=345851,783755,200789
BC00603=345851,783755,200789
BC00604=345851,783755,200789
BC00605=345851,783755,200789
BC00606=345851,783755,200789
BC00607=345851,783755,200789
BC00608=345851,783755,200789
BC00609=345851,783755,200789
BC00610=345851,783755,200789
BC00611=345851,783755,200789
BC00612=345851,783755,200789
BC00613=319787,789553,203514
BC00614=319787,789553,203514
BC00615=319787,789553,203514
BC00616=319787,789553,203514
BC00617=319787,789553,203514
BC00618=319787,789553,203514
BC00619=319787,789553,203514
BC00620=319787,789553,203514
BC00621=319787,789553,203514
BC00622=359964,789553,203647
BC00623=359964,789553,203647
BC00624=359964,789553,203647
BC00625=359964,789553,203647
BC00626=359964,789553,203647
BC00627=359964,789553,203647
BC00628=359964,789553,203647
BC00629=359964,789553,203647
BC00630=359964,789553,203647
BC00631=359964,789553,203647
BC00632=365235,789553,136516
BC00633=365235,789553,136516
BC00634=365235,789553,136516
BC00635=365235,789553,136516
BC00636=365235,789553,136516
BC00637=365235,789553,136516
BC00638=365234,789553,136512
BC00639=365234,789553,136512
BC00640=365234,789553,136512
BC00641=365235,789553,136516
BC00642=365235,789553,136516
BC00643=365235,669876,311777
BC00644=219200,669876,311777
BC00645=202290,739783,276486
BC00646=196160,765124,263693
BC00647=196160,765124,263693
BC00648=196160,765124,263693
BC00649=196160,765124,263693
BC00650=196160,765124,263693
BC00651=196160,765124,263693
BC00652=196160,765124,263693
BC00653=196160,765124,263693
BC00654=196160,765124,263693
BC00655=196160,765124,263693
BC00656=179300,757654,148443
BC00657=179300,757654,148443
BC00658=179300,757654,148443
BC00659=179300,757654,148443
BC00660=179301,757656,148440
BC00661=179301,757656,148440
BC00662=179301,757656,148440
BC00663=179301,757656,148440
BC00664=179301,757656,148440
BC00665=179300,757654,148443
BC00666=202290,739783,276486
BC00667=219200,669876,311777
BC00668=365235,669876,311777
BC00669=365235,789553,136516
BC00670=312307,789553,228155
BC00671=312307,789553,228155
BC00672=312307,789553,228155
BC00673=312307,789553,228155
BC00674=312307,789553,228155
BC00675=312307,789553,228155
BC00676=312307,789553,228155
BC00677=312307,789553,228155
BC00678=312307,789553,228155
BC00679=312307,789553,228155
BC00680=312307,789553,228155
BC00681=312307,789553,228155
BC00682=312307,789553,228155
BC00683=312307,789553,228155
BC00684=312307,789553,228155
BC00685=312307,789553,228155
BC00686=312307,789553,228155
BC00687=315278,774952,138157
BC00688=315278,774952,138157
BC00689=315278,774952,138157
BC00690=315278,774952,138157
BC00691=315278,774952,138157
BC00692=315278,774952,138157
BC00693=315278,774952,138157
BC00694=349744,788873,128099
BC00695=349744,788873,128099
BC00696=349744,788873,128099
BC00697=349744,788873,128099
BC00698=349744,788873,128099
BC00699=349744,788873,128099
BC00700=349744,788873,128099
BC00701=382626,789553,75740
BC00702=382626,789553,75740
BC00703=382625,789552,75737
BC00704=382625,789552,75737
BC00705=382626,789553,75740
BC00706=382626,789553,75740
BC00707=357624,789553,120797
BC00708=357624,789553,120797
BC00709=357624,789553,120797
BC00710=356987,789553,120797
BC00711=357624,789553,120797
BC00712=357624,789553,120797
BC00713=322012,789553,130156
BC00714=296072,789553,136973
BC00715=296072,789553,136973
BC00716=296072,789553,136973
BC00717=296072,789553,136973
BC00718=296072,789553,136973
BC00719=296072,789553,136973
BC00720=317007,789553,149819
BC00721=317007,789553,149819
BC00722=317007,789553,149819
BC00723=317007,789553,149819
BC00724=317007,789553,149819
BC00725=317007,789553,149819
BC00726=322972,789553,141208
BC00727=322972,789553,141208
BC00728=322972,789553,141208
BC00729=322972,789553,141208
BC00730=322972,789553,141208
BC00731=322972,789553,141208
BC00732=322972,668461,141208
BC00733=182890,668461,141208
BC00734=138897,773188,238096
BC00735=138897,773188,238096
BC00736=138897,773188,238096
BC00737=138897,773188,238096
BC00738=138897,773188,238096
BC00739=138897,773188,238096
BC00740=210738,761007,251818
BC00741=210738,761007,251818
BC00742=210738,761007,251818
BC00743=210738,761007,251818
BC00744=210738,761007,251818
BC00745=210738,761007,251818
BC00746=187715,774579,182649
BC00747=187715,774579,182649
BC00748=187715,774579,182649
BC00749=187715,774579,182649
BC00750=187715,774579,182649
BC00751=187715,774579,182649
BC00752=187905,774497,182612
BC00753=187905,774497,182612
BC00754=187905,774497,182612
BC00755=187905,774497,182612
BC00756=187905,774497,182612
BC00757=187905,774497,182612
BC00758=182890,668461,141208
BC00759=322972,668461,141208
BC00760=380287,789553,141173
BC00761=380287,789553,141173
BC00762=380287,789553,141173
BC00763=380287,789553,141173
BC00764=380287,789553,141173
BC00765=380287,789553,141173
BC00766=371434,789553,120731
BC00767=371434,789553,120731
BC00768=371434,789553,120731
BC00769=371434,789553,120731
BC00770=371434,789553,120731
BC00771=371434,789553,120731
BC00772=371434,685314,120731
BC00773=165820,667836,534036
EC00000=798156,0
EC00001=798156,0
EC00002=798156,0
EC00003=798156,0
EC00004=798156,0
EC00005=798156,0
EC00006=798156,0
EC00007=798156,0
EC00008=798156,0
EC00009=798156,0
EC00010=798156,0
EC00011=798156,0
EC00012=798156,0
EC00013=798156,0
EC00014=798156,0
EC00015=798156,0
EC00016=798156,0
EC00017=798156,0
EC00018=798156,0
EC00019=798156,0
EC00020=798156,0
EC00021=798156,0
EC00022=798156,0
EC00023=798156,0
EC00024=798156,0
EC00025=798156,0
EC00026=798156,0
EC00027=798156,0
EC00028=798156,0
EC00029=798156,0
EC00030=798156,0
EC00031=798156,0
EC00032=798156,0
EC00033=798156,0
EC00034=798156,0
EC00035=798156,0
EC00036=798156,0
EC00037=798156,0
EC00038=798156,0
EC00039=798156,0
EC00040=798156,0
EC00041=798156,0
EC00042=798156,0
EC00043=798156,0
EC00044=798156,0
EC00045=798156,0
EC00046=798156,0
EC00047=798156,0
EC00048=798156,0
EC00049=798156,0
EC00050=798156,0
EC00051=798156,0
EC00052=798156,0
EC00053=798156,0
EC00054=798156,0
EC00055=798156,0
EC00056=798156,0
EC00057=798156,0
EC00058=798156,0
EC00059=798156,0
EC00060=798156,0
EC00061=798156,0
EC00062=798156,0
EC00063=798156,0
EC00064=798156,0
EC00065=798156,0
EC00066=798156,0
EC00067=798156,0
EC00068=798156,0
EC00069=798156,0
EC00070=798156,0
EC00071=798156,0
EC00072=798156,0
EC00073=798156,0
EC00074=798156,0
EC00075=798156,0
EC00076=798156,0
EC00077=798156,0
EC00078=798156,0
EC00079=798156,0
EC00080=798156,0
EC00081=798156,0
EC00082=798156,0
EC00083=798156,0
EC00084=798156,0
EC00085=798156,0
EC00086=798156,0
EC00087=798156,0
EC00088=798156,0
EC00089=798156,0
EC00090=798156,0
EC00091=798156,0
EC00092=798156,0
EC00093=798156,0
EC00094=798156,0
EC00095=798156,0
EC00096=798156,0
EC00097=798156,0
EC00098=798156,0
EC00099=798156,0
EC00100=798156,0
EC00101=798156,0
EC00102=798156,0
EC00103=798156,0
EC00104=798156,0
EC00105=798156,0
EC00106=798156,0
EC00107=798156,0
EC00108=798156,0
EC00109=798156,0
EC00110=798156,0
EC00111=798156,0
EC00112=798156,0
EC00113=798156,0
EC00114=798156,0
EC00115=798156,0
EC00116=798156,0
EC00117=798156,0
EC00118=798156,0
EC00119=798156,0
EC00120=798156,0
EC00121=798156,0
EC00122=798156,0
EC00123=798156,0
EC00124=798156,0
EC00125=798156,0
EC00126=798156,0
EC00127=798156,0
EC00128=798156,0
EC00129=798156,0
EC00130=798156,0
EC00131=798156,0
EC00132=798156,0
EC00133=798156,0
EC00134=798156,0
EC00135=798156,0
EC00136=798156,0
EC00137=798156,0
EC00138=798156,0
EC00139=798156,0
EC00140=798156,0
EC00141=798156,0
EC00142=798156,0
EC00143=798156,0
EC00144=798156,0
EC00145=798156,0
EC00146=798156,0
EC00147=798156,0
EC00148=798156,0
EC00149=798156,0
EC00150=798156,0
EC00151=798156,0
EC00152=798156,0
EC00153=798156,0
EC00154=798156,0
EC00155=798156,0
EC00156=798156,0
EC00157=798156,0
EC00158=798156,0
EC00159=798156,0
EC00160=798156,0
EC00161=798156,0
EC00162=798156,0
EC00163=798156,0
EC00164=798156,0
EC00165=798156,0
EC00166=798156,0
EC00167=798156,0
EC00168=798156,0
EC00169=798156,0
EC00170=798156,0
EC00171=798156,0
EC00172=798156,0
EC00173=798155,0
EC00174=798155,1
EC00175=798155,0
EC00176=798155,1
EC00177=798156,0
EC00178=798156,0
EC00179=798156,0
EC00180=798156,0
EC00181=798156,0
EC00182=798156,0
EC00183=798156,0
EC00184=798156,0
EC00185=798156,0
EC00186=798156,0
EC00187=798156,0
EC00188=798156,0
EC00189=798156,0
EC00190=798156,0
EC00191=798156,0
EC00192=798156,0
EC00193=798153,3
EC00194=798156,0
EC00195=798156,0
EC00196=798156,0
EC00197=798156,0
EC00198=798156,0
EC00199=798156,0
EC00200=798156,0
EC00201=798156,0
EC00202=798156,0
EC00203=798156,0
EC00204=798156,0
EC00205=798156,0
EC00206=798155,0
EC00207=798156,0
EC00208=798156,0
EC00209=798156,0
EC00210=798156,0
EC00211=798156,0
EC00212=798156,0
EC00213=798156,0
EC00214=798156,0
EC00215=798156,0
EC00216=798156,0
EC00217=798156,0
EC00218=798156,0
EC00219=798156,0
EC00220=798156,0
EC00221=798156,0
EC00222=798156,0
EC00223=798156,0
EC00224=798155,1
EC00225=798155,1
EC00226=798155,0
EC00227=798156,0
EC00228=798156,0
EC00229=798156,0
EC00230=798156,0
EC00231=798156,0
EC00232=798156,0
EC00233=798156,0
EC00234=798156,0
EC00235=798156,0
EC00236=798156,0
EC00237=798156,0
EC00238=798156,0
EC00239=798156,0
EC00240=798156,0
EC00241=798156,0
EC00242=798156,0
EC00243=798156,0
EC00244=798156,0
EC00245=798156,0
EC00246=798156,0
EC00247=798156,0
EC00248=798156,0
EC00249=798155,0
EC00250=798156,0
EC00251=798156,0
EC00252=798156,0
EC00253=798156,0
EC00254=798156,0
EC00255=798156,0
EC00256=798156,0
EC00257=798156,0
EC00258=798156,0
EC00259=798156,0
EC00260=798156,0
EC00261=798156,0
EC00262=798156,0
EC00263=798156,0
EC00264=798156,0
EC00265=798156,0
EC00266=798156,0
EC00267=798156,0
EC00268=798156,0
EC00269=798156,0
EC00270=798156,0
EC00271=798156,0
EC00272=798156,0
EC00273=798156,0
EC00274=798156,0
EC00275=798156,0
EC00276=798156,0
EC00277=798156,0
EC00278=798156,0
EC00279=798156,0
EC00280=798156,0
EC00281=798156,0
EC00282=798156,0
EC00283=798156,0
EC00284=798156,0
EC00285=798156,0
EC00286=798156,0
EC00287=798156,0
EC00288=798156,0
EC00289=798156,0
EC00290=798156,0
EC00291=798156,0
EC00292=798156,0
EC00293=798156,0
EC00294=798156,0
EC00295=798156,0
EC00296=798156,0
EC00297=798156,0
EC00298=798156,0
EC00299=798156,0
EC00300=798156,0
EC00301=798156,0
EC00302=798156,0
EC00303=798156,0
EC00304=798156,0
EC00305=798156,0
EC00306=798156,0
EC00307=798156,0
EC00308=798156,0
EC00309=798156,0
EC00310=798156,0
EC00311=798156,0
EC00312=798156,0
EC00313=798156,0
EC00314=798156,0
EC00315=798156,0
EC00316=798156,0
EC00317=798156,0
EC00318=798156,0
EC00319=798156,0
EC00320=798156,0
EC00321=798156,0
EC00322=798156,0
EC00323=798156,0
EC00324=798156,0
EC00325=798156,0
EC00326=798156,0
EC00327=798156,0
EC00328=798156,0
EC00329=798156,0
EC00330=798156,0
EC00331=798156,0
EC00332=798156,0
EC00333=798156,0
EC00334=798156,0
EC00335=798156,0
EC00336=798156,0
EC00337=798156,0
EC00338=798156,0
EC00339=798156,0
EC00340=798156,0
EC00341=798156,0
EC00342=798156,0
EC00343=798156,0
EC00344=798156,0
EC00345=798156,0
EC00346=798156,0
EC00347=798156,0
EC00348=798156,0
EC00349=798156,0
EC00350=798156,0
EC00351=798156,0
EC00352=798156,0
EC00353=798156,0
EC00354=798156,0
EC00355=798156,0
EC00356=798156,0
EC00357=798156,0
EC00358=798156,0
EC00359=798156,0
EC00360=798156,0
EC00361=798156,0
EC00362=798156,0
EC00363=798156,0
EC00364=798156,0
EC00365=798156,0
EC00366=798156,0
EC00367=798156,0
EC00368=798156,0
EC00369=798156,0
EC00370=798156,0
EC00371=798156,0
EC00372=798156,0
EC00373=798156,0
EC00374=798156,0
EC00375=798156,0
EC00376=798156,0
EC00377=798156,0
EC00378=798156,0
EC00379=798156,0
EC00380=798156,0
EC00381=798156,0
EC00382=798156,0
EC00383=798156,0
EC00384=798156,0
EC00385=798156,0
EC00386=798156,0
EC00387=798156,0
EC00388=798156,0
EC00389=798156,0
EC00390=798156,0
EC00391=798156,0
EC00392=798156,0
EC00393=798156,0
EC00394=798156,0
EC00395=798156,0
EC00396=798156,0
EC00397=798156,0
EC00398=798156,0
EC00399=798156,0
EC00400=798156,0
EC00401=798156,0
EC00402=798156,0
EC00403=798156,0
EC00404=798156,0
EC00405=798156,0
EC00406=798156,0
EC00407=798156,0
EC00408=798156,0
EC00409=798156,0
EC00410=798156,0
EC00411=798156,0
EC00412=798156,0
EC00413=798156,0
EC00414=798156,0
EC00415=798156,0
EC00416=798156,0
EC00417=798156,0
EC00418=798156,0
EC00419=798156,0
EC00420=798156,0
EC00421=798156,0
EC00422=798156,0
EC00423=798156,0
EC00424=798156,0
EC00425=798156,0
EC00426=798156,0
EC00427=798156,0
EC00428=798156,0
EC00429=798156,0
EC00430=798156,0
EC00431=798156,0
EC00432=798156,0
EC00433=798156,0
EC00434=798156,0
EC00435=798156,0
EC00436=798156,0
EC00437=798156,0
EC00438=798156,0
EC00439=798156,0
EC00440=798156,0
EC00441=798156,0
EC00442=798156,0
EC00443=798156,0
EC00444=798156,0
EC00445=798156,0
EC00446=798156,0
EC00447=798156,0
EC00448=798156,0
EC00449=798156,0
EC00450=798156,0
EC00451=798155,0
EC00452=798155,1
EC00453=798155,0
EC00454=798155,1
EC00455=798156,0
EC00456=798156,0
EC00457=798156,0
EC00458=798156,0
EC00459=798156,0
EC00460=798156,0
EC00461=798156,0
EC00462=798156,0
EC00463=798156,0
EC00464=798156,0
EC00465=798156,0
EC00466=798156,0
EC00467=798156,0
EC00468=798156,0
EC00469=798156,0
EC00470=798156,0
EC00471=798153,3
EC00472=798156,0
EC00473=798156,0
EC00474=798156,0
EC00475=798156,0
EC00476=798156,0
EC00477=798156,0
EC00478=798156,0
EC00479=798156,0
EC00480=798156,0
EC00481=798156,0
EC00482=798156,0
EC00483=798156,0
EC00484=798155,0
EC00485=798156,0
EC00486=798156,0
EC00487=798156,0
EC00488=798156,0
EC00489=798156,0
EC00490=798156,0
EC00491=798156,0
EC00492=798156,0
EC00493=798156,0
EC00494=798156,0
EC00495=798156,0
EC00496=798156,0
EC00497=798156,0
EC00498=798156,0
EC00499=798156,0
EC00500=798156,0
EC00501=798156,0
EC00502=798156,0
EC00503=798156,0
EC00504=798155,0
EC00505=798156,0
EC00506=798156,0
EC00507=798156,0
EC00508=798156,0
EC00509=798156,0
EC00510=798156,0
EC00511=798156,0
EC00512=798156,0
EC00513=798156,0
EC00514=798156,0
EC00515=798156,0
EC00516=798156,0
EC00517=798156,0
EC00518=798156,0
EC00519=798156,0
EC00520=798156,0
EC00521=798156,0
EC00522=798156,0
EC00523=798156,0
EC00524=798156,0
EC00525=798156,0
EC00526=798156,0
EC00527=798155,0
EC00528=798156,0
EC00529=798156,0
EC00530=798156,0
EC00531=798156,0
EC00532=798156,0
EC00533=798156,0
EC00534=798156,0
EC00535=798156,0
EC00536=798156,0
EC00537=798156,0
EC00538=798156,0
EC00539=798156,0
EC00540=798156,0
EC00541=798156,0
EC00542=798156,0
EC00543=798156,0
EC00544=798156,0
EC00545=798156,0
EC00546=798156,0
EC00547=798156,0
EC00548=798156,0
EC00549=798156,0
EC00550=798156,0
EC00551=798156,0
EC00552=798156,0
EC00553=798156,0
EC00554=798156,0
EC00555=798156,0
EC00556=798156,0
EC00557=798156,0
EC00558=798156,0
EC00559=798156,0
EC00560=798156,0
EC00561=798156,0
EC00562=798156,0
EC00563=798156,0
EC00564=798156,0
EC00565=798156,0
EC00566=798156,0
EC00567=798156,0
EC00568=798156,0
EC00569=798156,0
EC00570=798156,0
EC00571=798156,0
EC00572=798156,0
EC00573=798156,0
EC00574=798156,0
EC00575=798156,0
EC00576=798156,0
EC00577=798156,0
EC00578=798156,0
EC00579=798156,0
EC00580=798156,0
EC00581=798156,0
EC00582=798156,0
EC00583=798156,0
EC00584=798156,0
EC00585=798156,0
EC00586=798156,0
EC00587=798156,0
EC00588=798156,0
EC00589=798156,0
EC00590=798156,0
EC00591=798156,0
EC00592=798156,0
EC00593=798156,0
EC00594=798156,0
EC00595=798156,0
EC00596=798156,0
EC00597=798156,0
EC00598=798156,0
EC00599=798156,0
EC00600=798156,0
EC00601=798156,0
EC00602=798156,0
EC00603=798156,0
EC00604=798156,0
EC00605=798156,0
EC00606=798156,0
EC00607=798156,0
EC00608=798156,0
EC00609=798156,0
EC00610=798156,0
EC00611=798156,0
EC00612=798156,0
EC00613=798156,0
EC00614=798156,0
EC00615=798156,0
EC00616=798156,0
EC00617=798156,0
EC00618=798156,0
EC00619=798156,0
EC00620=798156,0
EC00621=798156,0
EC00622=798156,0
EC00623=798156,0
EC00624=798156,0
EC00625=798156,0
EC00626=798156,0
EC00627=798156,0
EC00628=798156,0
EC00629=798156,0
EC00630=798156,0
EC00631=798156,0
EC00632=798156,0
EC00633=798156,0
EC00634=798156,0
EC00635=798156,0
EC00636=798156,0
EC00637=798156,0
EC00638=798155,0
EC00639=798155,0
EC00640=798155,0
EC00641=798156,0
EC00642=798156,0
EC00643=798156,0
EC00644=798156,0
EC00645=798156,0
EC00646=798156,0
EC00647=798156,0
EC00648=798156,0
EC00649=798156,0
EC00650=798156,0
EC00651=798156,0
EC00652=798156,0
EC00653=798156,0
EC00654=798156,0
EC00655=798156,0
EC00656=798156,0
EC00657=798156,0
EC00658=798156,0
EC00659=798156,0
EC00660=798155,0
EC00661=798155,0
EC00662=798155,0
EC00663=798155,0
EC00664=798155,0
EC00665=798156,0
EC00666=798156,0
EC00667=798156,0
EC00668=798156,0
EC00669=798156,0
EC00670=798156,0
EC00671=798156,0
EC00672=798156,0
EC00673=798156,0
EC00674=798156,0
EC00675=798156,0
EC00676=798156,0
EC00677=798156,0
EC00678=798156,0
EC00679=798156,0
EC00680=798156,0
EC00681=798156,0
EC00682=798156,0
EC00683=798156,0
EC00684=798156,0
EC00685=798156,0
EC00686=798156,0
EC00687=798156,0
EC00688=798156,0
EC00689=798156,0
EC00690=798156,0
EC00691=798156,0
EC00692=798156,0
EC00693=798156,0
EC00694=798156,0
EC00695=798156,0
EC00696=798156,0
EC00697=798156,0
EC00698=798156,0
EC00699=798156,0
EC00700=798156,0
EC00701=798156,0
EC00702=798156,0
EC00703=798155,0
EC00704=798155,0
EC00705=798156,0
EC00706=798156,0
EC00707=798156,0
EC00708=798156,0
EC00709=798156,0
EC00710=798156,0
EC00711=798156,0
EC00712=798156,0
EC00713=798156,0
EC00714=798156,0
EC00715=798156,0
EC00716=798156,0
EC00717=798156,0
EC00718=798156,0
EC00719=798156,0
EC00720=798156,0
EC00721=798156,0
EC00722=798156,0
EC00723=798156,0
EC00724=798156,0
EC00725=798156,0
EC00726=798156,0
EC00727=798156,0
EC00728=798156,0
EC00729=798156,0
EC00730=798156,0
EC00731=798156,0
EC00732=798156,0
EC00733=798156,0
EC00734=798156,0
EC00735=798156,0
EC00736=798156,0
EC00737=798156,0
EC00738=798156,0
EC00739=798156,0
EC00740=798156,0
EC00741=798156,0
EC00742=798156,0
EC00743=798156,0
EC00744=798156,0
EC00745=798156,0
EC00746=798156,0
EC00747=798156,0
EC00748=798156,0
EC00749=798156,0
EC00750=798156,0
EC00751=798156,0
EC00752=798156,0
EC00753=798156,0
EC00754=798156,0
EC00755=798156,0
EC00756=798156,0
EC00757=798156,0
EC00758=798156,0
EC00759=798156,0
EC00760=798156,0
EC00761=798156,0
EC00762=798156,0
EC00763=798156,0
EC00764=798156,0
EC00765=798156,0
EC00766=798156,0
EC00767=798156,0
EC00768=798156,0
EC00769=798156,0
EC00770=798156,0
EC00771=798156,0
EC00772=798156,0
EC00773=798156,0
///POSTYPE BASE
///RECTAN
///RCONF 0,0,0,0,0,0,0,0,0,0,0,0,0,0,0,0,0,0,0,0,0,0,0,0
P00006=0.222,-3.123,-1.508,0.0000,0.0000,0.0000
P00021=-0.225,-6.128,-0.405,0.0000,0.0000,0.0000
P00022=0.222,-3.123,-1.508,0.0000,0.0000,0.0000
P00023=0.143,-0.036,0.682,0.0000,0.0000,0.0000
P00024=0.145,-0.552,1.326,0.0000,0.0000,0.0000
P00025=-2.003,0.006,0.728,0.0000,0.0000,0.0000
P00026=0.562,-0.002,-0.337,0.0000,0.0000,0.0000
P00027=-0.746,0.015,-9.096,0.0000,0.0000,0.0000
P00028=-2.237,-0.018,-7.702,0.0000,0.0000,0.0000
P00029=-2.156,-0.086,-4.681,0.0000,0.0000,0.0000
P00030=5.926,-4.294,-1.390,0.0000,0.0000,0.0000
P00031=1.853,-0.001,-1.549,0.0000,0.0000,0.0000
P00032=1.957,0.503,-7.217,0.0000,0.0000,0.0000
///RCONF 0,0,0,0,1,0,0,0,0,0,0,0,0,0,0,0,0,0,0,0,0,0,0,0
P00033=-0.123,0.612,-5.012,0.0000,0.0000,0.0000
///RCONF 0,0,0,0,0,0,0,0,0,0,0,0,0,0,0,0,0,0,0,0,0,0,0,0
P00034=-0.304,0.773,-2.693,0.0000,0.0000,0.0000
P00042=-0.217,1.941,0.413,0.0000,0.0000,0.0000
P00043=-0.044,-1.937,1.197,0.0000,0.0000,0.0000
P00044=0.687,-2.322,1.156,0.0000,0.0000,0.0000
P00045=-0.068,-0.810,1.603,0.0000,0.0000,0.0000
P00046=0.799,0.043,1.292,0.0000,0.0000,0.0000
///RCONF 0,1,0,0,0,0,0,0,0,0,0,0,0,0,0,0,0,0,0,0,0,0,0,0
P00047=-0.011,1.737,-0.646,0.0000,0.0000,0.0000
///RCONF 0,0,0,0,0,0,0,0,0,0,0,0,0,0,0,0,0,0,0,0,0,0,0,0
P00048=2.411,0.025,-0.606,0.0000,0.0000,0.0000
P00049=3.413,-3.572,-1.618,0.0000,0.0000,0.0000
P00050=4.296,-4.501,-0.826,0.0000,0.0000,0.0000
P00051=0.367,3.892,0.009,0.0000,0.0000,0.0000
P00060=2.327,-2.514,-2.692,0.0000,0.0000,0.0000
P00091=-0.109,0.052,-0.075,0.0000,0.0000,0.0000
//INST
///DATE 2025/03/12 10:33
///ATTR SC,RW
///GROUP1 RB1,BS1
///GROUP2 ST1
NOP
COMM 'X2_38-47,64(2)(90,0)
COMM 'Down
COMM MOVJ C00000 BC00000 VJ=100.00  +MOVJ EC00000 VJ=100.00
COMM 'Up
COMM 'Path S4602
COMM SFTOF3D
COMM MOVJ C00001 BC00001 VJ=100.00  +MOVJ EC00001 VJ=100.00
COMM MOVL C00002 BC00002 V=800.0  +MOVJ EC00002 VJ=100.00
COMM SMOVL C00003 BC00003 V=166.7  +MOVJ EC00003
COMM SREFP 3 C00004 BC00004  +REFP EC00004
COMM CALL JOB:SEARCH-R1-S13D
COMM SET P021 P006
COMM SFTON3D P021
COMM SMOVL C00005 BC00005 V=166.7  +MOVJ EC00005
COMM SREFP 3 C00006 BC00006  +REFP EC00006
COMM CALL JOB:SEARCH-R1-S13D
COMM SET P021 P006
COMM SFTON3D P021
COMM SMOVL C00007 BC00007 V=166.7  +MOVJ EC00007
COMM MOVL C00008 BC00008 V=1000.0  +MOVJ EC00008 VJ=100.00
COMM 'EndPath S4602
COMM 'Path S4603
COMM SFTOF3D
COMM MOVJ C00009 BC00009 VJ=100.00  +MOVJ EC00009 VJ=100.00
COMM MOVL C00010 BC00010 V=800.0  +MOVJ EC00010 VJ=100.00
COMM SMOVL C00011 BC00011 V=166.7  +MOVJ EC00011
COMM SREFP 3 C00012 BC00012  +REFP EC00012
COMM CALL JOB:SEARCH-R1-S13D
COMM SET P022 P006
COMM SFTON3D P022
COMM SMOVL C00013 BC00013 V=166.7  +MOVJ EC00013
COMM SREFP 3 C00014 BC00014  +REFP EC00014
COMM CALL JOB:SEARCH-R1-S13D
COMM SET P022 P006
COMM SFTON3D P022
COMM SMOVL C00015 BC00015 V=166.7  +MOVJ EC00015
COMM MOVL C00016 BC00016 V=1000.0  +MOVJ EC00016 VJ=100.00
COMM 'EndPath S4603
COMM 'Path S4604
COMM SFTOF3D
COMM MOVJ C00017 BC00017 VJ=100.00  +MOVJ EC00017 VJ=100.00
COMM MOVJ C00018 BC00018 VJ=100.00  +MOVJ EC00018 VJ=100.00
COMM MOVL C00019 BC00019 V=800.0  +MOVJ EC00019 VJ=100.00
COMM SMOVL C00020 BC00020 V=166.7  +MOVJ EC00020
COMM SREFP 3 C00021 BC00021  +REFP EC00021
COMM CALL JOB:SEARCH-R1-S13D
COMM SET P023 P006
COMM SFTON3D P023
COMM SMOVL C00022 BC00022 V=166.7  +MOVJ EC00022
COMM SREFP 3 C00023 BC00023  +REFP EC00023
COMM CALL JOB:SEARCH-R1-S13D
COMM SET P023 P006
COMM SFTON3D P023
COMM SMOVL C00024 BC00024 V=166.7  +MOVJ EC00024
COMM SMOVL C00025 BC00025 V=333.3  +MOVJ EC00025
COMM SMOVL C00026 BC00026 V=333.3  +MOVJ EC00026
COMM SREFP 3 C00027 BC00027  +REFP EC00027
COMM CALL JOB:SEARCH-R1-S13D
COMM SET P023 P006
COMM SFTON3D P023
COMM SMOVL C00028 BC00028 V=166.7  +MOVJ EC00028
COMM MOVL C00029 BC00029 V=1000.0  +MOVJ EC00029 VJ=100.00
COMM 'EndPath S4604
COMM 'Path S4605
COMM SFTOF3D
COMM MOVJ C00030 BC00030 VJ=100.00  +MOVJ EC00030 VJ=100.00
COMM MOVL C00031 BC00031 V=800.0  +MOVJ EC00031 VJ=100.00
COMM SMOVL C00032 BC00032 V=166.7  +MOVJ EC00032
COMM SREFP 3 C00033 BC00033  +REFP EC00033
COMM CALL JOB:SEARCH-R1-S13D
COMM SET P024 P006
COMM SFTON3D P024
COMM SMOVL C00034 BC00034 V=166.7  +MOVJ EC00034
COMM SMOVL C00035 BC00035 V=166.7  +MOVJ EC00035
COMM SREFP 3 C00036 BC00036  +REFP EC00036
COMM CALL JOB:SEARCH-R1-S13D
COMM SET P024 P006
COMM SFTON3D P024
COMM SMOVL C00037 BC00037 V=166.7  +MOVJ EC00037
COMM SMOVL C00038 BC00038 V=166.7  +MOVJ EC00038
COMM SREFP 3 C00039 BC00039  +REFP EC00039
COMM CALL JOB:SEARCH-R1-S13D
COMM SET P024 P006
COMM SFTON3D P024
COMM SMOVL C00040 BC00040 V=166.7  +MOVJ EC00040
COMM MOVL C00041 BC00041 V=1000.0  +MOVJ EC00041 VJ=100.00
COMM MOVL C00042 BC00042 V=1000.0  +MOVJ EC00042 VJ=100.00
COMM 'EndPath S4605
COMM 'Path S4606
COMM SFTOF3D
COMM MOVJ C00043 BC00043 VJ=100.00  +MOVJ EC00043 VJ=100.00
COMM MOVL C00044 BC00044 V=800.0  +MOVJ EC00044 VJ=100.00
COMM SMOVL C00045 BC00045 V=166.7  +MOVJ EC00045
COMM SREFP 3 C00046 BC00046  +REFP EC00046
COMM CALL JOB:SEARCH-R1-S13D
COMM SET P025 P006
COMM SFTON3D P025
COMM SMOVL C00047 BC00047 V=166.7  +MOVJ EC00047
COMM SREFP 3 C00048 BC00048  +REFP EC00048
COMM CALL JOB:SEARCH-R1-S13D
COMM SET P025 P006
COMM SFTON3D P025
COMM SMOVL C00049 BC00049 V=166.7  +MOVJ EC00049
COMM SMOVL C00050 BC00050 V=166.7  +MOVJ EC00050
COMM SREFP 3 C00051 BC00051  +REFP EC00051
COMM CALL JOB:SEARCH-R1-S13D
COMM SET P025 P006
COMM SFTON3D P025
COMM SMOVL C00052 BC00052 V=166.7  +MOVJ EC00052
COMM MOVL C00053 BC00053 V=1000.0  +MOVJ EC00053 VJ=100.00
COMM MOVL C00054 BC00054 V=1000.0  +MOVJ EC00054 VJ=100.00
COMM 'EndPath S4606
COMM 'Path S4607
COMM SFTOF3D
COMM MOVJ C00055 BC00055 VJ=100.00  +MOVJ EC00055 VJ=100.00
COMM MOVL C00056 BC00056 V=800.0  +MOVJ EC00056 VJ=100.00
COMM SMOVL C00057 BC00057 V=166.7  +MOVJ EC00057
COMM SREFP 3 C00058 BC00058  +REFP EC00058
COMM CALL JOB:SEARCH-R1-S13D
COMM SET P026 P006
COMM SFTON3D P026
COMM SMOVL C00059 BC00059 V=166.7  +MOVJ EC00059
COMM SREFP 3 C00060 BC00060  +REFP EC00060
COMM CALL JOB:SEARCH-R1-S13D
COMM SET P026 P006
COMM SFTON3D P026
COMM SMOVL C00061 BC00061 V=166.7  +MOVJ EC00061
COMM MOVL C00062 BC00062 V=1000.0  +MOVJ EC00062 VJ=100.00
COMM SFTOF3D
COMM SMOVL C00063 BC00063 V=166.7  +MOVJ EC00063
COMM SREFP 3 C00064 BC00064  +REFP EC00064
COMM CALL JOB:SEARCH-R1-S13D
COMM SET P091 P006
COMM SFTON3D P091
COMM SMOVL C00065 BC00065 V=166.7  +MOVJ EC00065
COMM SREFP 3 C00066 BC00066  +REFP EC00066
COMM CALL JOB:SEARCH-R1-S13D
COMM SET P091 P006
COMM SFTON3D P091
COMM SMOVL C00067 BC00067 V=166.7  +MOVJ EC00067
COMM SMOVL C00068 BC00068 V=500.0  +MOVJ EC00068
COMM 'EndPath S4607
COMM MOVJ C00069 BC00069 VJ=100.00  +MOVJ EC00069 VJ=100.00
COMM MOVJ C00070 BC00070 VJ=100.00  +MOVJ EC00070 VJ=100.00
COMM 'Path S4608
COMM SFTOF3D
COMM MOVJ C00071 BC00071 VJ=100.00  +MOVJ EC00071 VJ=100.00
COMM MOVL C00072 BC00072 V=800.0  +MOVJ EC00072 VJ=100.00
COMM SMOVL C00073 BC00073 V=166.7  +MOVJ EC00073
COMM SREFP 3 C00074 BC00074  +REFP EC00074
COMM CALL JOB:SEARCH-R1-S13D
COMM SET P027 P006
COMM SFTON3D P027
COMM SMOVL C00075 BC00075 V=166.7  +MOVJ EC00075
COMM SMOVL C00076 BC00076 V=166.7  +MOVJ EC00076
COMM SREFP 3 C00077 BC00077  +REFP EC00077
COMM CALL JOB:SEARCH-R1-S13D
COMM SET P027 P006
COMM SFTON3D P027
COMM SMOVL C00078 BC00078 V=166.7  +MOVJ EC00078
COMM SMOVL C00079 BC00079 V=166.7  +MOVJ EC00079
COMM SREFP 3 C00080 BC00080  +REFP EC00080
COMM CALL JOB:SEARCH-R1-S13D
COMM SET P027 P006
COMM SFTON3D P027
COMM SMOVL C00081 BC00081 V=166.7  +MOVJ EC00081
COMM MOVL C00082 BC00082 V=1000.0  +MOVJ EC00082 VJ=100.00
COMM MOVL C00083 BC00083 V=1000.0  +MOVJ EC00083 VJ=100.00
COMM 'EndPath S4608
COMM 'Path S4609
COMM SFTOF3D
COMM MOVJ C00084 BC00084 VJ=100.00  +MOVJ EC00084 VJ=100.00
COMM MOVL C00085 BC00085 V=800.0  +MOVJ EC00085 VJ=100.00
COMM SMOVL C00086 BC00086 V=166.7  +MOVJ EC00086
COMM SREFP 3 C00087 BC00087  +REFP EC00087
COMM CALL JOB:SEARCH-R1-S13D
COMM SET P028 P006
COMM SFTON3D P028
COMM SMOVL C00088 BC00088 V=166.7  +MOVJ EC00088
COMM SREFP 3 C00089 BC00089  +REFP EC00089
COMM CALL JOB:SEARCH-R1-S13D
COMM SET P028 P006
COMM SFTON3D P028
COMM SMOVL C00090 BC00090 V=250.0  +MOVJ EC00090
COMM MOVL C00091 BC00091 V=1000.0  +MOVJ EC00091 VJ=100.00
COMM 'EndPath S4609
COMM MOVJ C00092 BC00092 VJ=100.00  +MOVJ EC00092 VJ=100.00
COMM 'Path S4882
COMM SFTOF3D
COMM MOVJ C00093 BC00093 VJ=100.00  +MOVJ EC00093 VJ=100.00
COMM MOVL C00094 BC00094 V=800.0  +MOVJ EC00094 VJ=100.00
COMM SMOVL C00095 BC00095 V=166.7  +MOVJ EC00095
COMM SREFP 3 C00096 BC00096  +REFP EC00096
COMM CALL JOB:SEARCH-R1-S13D
COMM SET P060 P006
COMM SFTON3D P060
COMM SMOVL C00097 BC00097 V=166.7  +MOVJ EC00097
COMM SMOVL C00098 BC00098 V=166.7  +MOVJ EC00098
COMM SREFP 3 C00099 BC00099  +REFP EC00099
COMM CALL JOB:SEARCH-R1-S13D
COMM SET P060 P006
COMM SFTON3D P060
COMM SMOVL C00100 BC00100 V=166.7  +MOVJ EC00100
COMM SMOVL C00101 BC00101 V=333.3  +MOVJ EC00101
COMM SMOVL C00102 BC00102 V=166.7  +MOVJ EC00102
COMM SREFP 3 C00103 BC00103  +REFP EC00103
COMM CALL JOB:SEARCH-R1-S13D
COMM SET P060 P006
COMM SFTON3D P060
COMM SMOVL C00104 BC00104 V=166.7  +MOVJ EC00104
COMM MOVL C00105 BC00105 V=1000.0  +MOVJ EC00105 VJ=100.00
COMM 'EndPath S4882
COMM MOVJ C00106 BC00106 VJ=100.00  +MOVJ EC00106 VJ=100.00
COMM 'Path S4610
COMM SFTOF3D
COMM MOVJ C00107 BC00107 VJ=100.00  +MOVJ EC00107 VJ=100.00
COMM MOVL C00108 BC00108 V=800.0  +MOVJ EC00108 VJ=100.00
COMM SMOVL C00109 BC00109 V=166.7  +MOVJ EC00109
COMM SREFP 3 C00110 BC00110  +REFP EC00110
COMM CALL JOB:SEARCH-R1-S13D
COMM SET P029 P006
COMM SFTON3D P029
COMM SMOVL C00111 BC00111 V=166.7  +MOVJ EC00111
COMM SREFP 3 C00112 BC00112  +REFP EC00112
COMM CALL JOB:SEARCH-R1-S13D
COMM SET P029 P006
COMM SFTON3D P029
COMM SMOVL C00113 BC00113 V=166.7  +MOVJ EC00113
COMM MOVL C00114 BC00114 V=1000.0  +MOVJ EC00114 VJ=100.00
COMM 'EndPath S4610
COMM 'Path S4611
COMM SFTOF3D
COMM MOVJ C00115 BC00115 VJ=100.00  +MOVJ EC00115 VJ=100.00
COMM MOVL C00116 BC00116 V=800.0  +MOVJ EC00116 VJ=100.00
COMM SMOVL C00117 BC00117 V=166.7  +MOVJ EC00117
COMM SREFP 3 C00118 BC00118  +REFP EC00118
COMM CALL JOB:SEARCH-R1-S13D
COMM SET P030 P006
COMM SFTON3D P030
COMM SMOVL C00119 BC00119 V=166.7  +MOVJ EC00119
COMM SREFP 3 C00120 BC00120  +REFP EC00120
COMM CALL JOB:SEARCH-R1-S13D
COMM SET P030 P006
COMM SFTON3D P030
COMM SMOVL C00121 BC00121 V=166.7  +MOVJ EC00121
COMM MOVL C00122 BC00122 V=800.0  +MOVJ EC00122 VJ=100.00
COMM MOVL C00123 BC00123 V=1000.0  +MOVJ EC00123 VJ=100.00
COMM 'EndPath S4611
COMM MOVJ C00124 BC00124 VJ=100.00  +MOVJ EC00124 VJ=100.00
COMM 'Path S4612
COMM SFTOF3D
COMM MOVJ C00125 BC00125 VJ=100.00  +MOVJ EC00125 VJ=100.00
COMM MOVL C00126 BC00126 V=800.0  +MOVJ EC00126 VJ=100.00
COMM SMOVL C00127 BC00127 V=166.7  +MOVJ EC00127
COMM SREFP 3 C00128 BC00128  +REFP EC00128
COMM CALL JOB:SEARCH-R1-S13D
COMM SET P031 P006
COMM SFTON3D P031
COMM SMOVL C00129 BC00129 V=166.7  +MOVJ EC00129
COMM SMOVL C00130 BC00130 V=166.7  +MOVJ EC00130
COMM SREFP 3 C00131 BC00131  +REFP EC00131
COMM CALL JOB:SEARCH-R1-S13D
COMM SET P031 P006
COMM SFTON3D P031
COMM SMOVL C00132 BC00132 V=166.7  +MOVJ EC00132
COMM SMOVL C00133 BC00133 V=166.7  +MOVJ EC00133
COMM SREFP 3 C00134 BC00134  +REFP EC00134
COMM CALL JOB:SEARCH-R1-S13D
COMM SET P031 P006
COMM SFTON3D P031
COMM SMOVL C00135 BC00135 V=166.7  +MOVJ EC00135
COMM MOVL C00136 BC00136 V=1000.0  +MOVJ EC00136 VJ=100.00
COMM 'EndPath S4612
COMM MOVJ C00137 BC00137 VJ=100.00  +MOVJ EC00137 VJ=100.00
COMM 'Path S4613
COMM SFTOF3D
COMM MOVJ C00138 BC00138 VJ=100.00  +MOVJ EC00138 VJ=100.00
COMM MOVL C00139 BC00139 V=800.0  +MOVJ EC00139 VJ=100.00
COMM SMOVL C00140 BC00140 V=166.7  +MOVJ EC00140
COMM SREFP 3 C00141 BC00141  +REFP EC00141
COMM CALL JOB:SEARCH-R1-S13D
COMM SET P032 P006
COMM SFTON3D P032
COMM SMOVL C00142 BC00142 V=166.7  +MOVJ EC00142
COMM SREFP 3 C00143 BC00143  +REFP EC00143
COMM CALL JOB:SEARCH-R1-S13D
COMM SET P032 P006
COMM SFTON3D P032
COMM SMOVL C00144 BC00144 V=166.7  +MOVJ EC00144
COMM SMOVL C00145 BC00145 V=166.7  +MOVJ EC00145
COMM SREFP 3 C00146 BC00146  +REFP EC00146
COMM CALL JOB:SEARCH-R1-S13D
COMM SET P032 P006
COMM SFTON3D P032
COMM SMOVL C00147 BC00147 V=166.7  +MOVJ EC00147
COMM MOVL C00148 BC00148 V=1000.0  +MOVJ EC00148 VJ=100.00
COMM 'EndPath S4613
COMM MOVJ C00149 BC00149 VJ=100.00  +MOVJ EC00149 VJ=100.00
COMM 'Path S4614
COMM SFTOF3D
COMM MOVJ C00150 BC00150 VJ=100.00  +MOVJ EC00150 VJ=100.00
COMM MOVL C00151 BC00151 V=800.0  +MOVJ EC00151 VJ=100.00
COMM SMOVL C00152 BC00152 V=166.7  +MOVJ EC00152
COMM SREFP 3 C00153 BC00153  +REFP EC00153
COMM CALL JOB:SEARCH-R1-S13D
COMM SET P033 P006
COMM SFTON3D P033
COMM SMOVL C00154 BC00154 V=166.7  +MOVJ EC00154
COMM SREFP 3 C00155 BC00155  +REFP EC00155
COMM CALL JOB:SEARCH-R1-S13D
COMM SET P033 P006
COMM SFTON3D P033
COMM SMOVL C00156 BC00156 V=166.7  +MOVJ EC00156
COMM MOVL C00157 BC00157 V=1000.0  +MOVJ EC00157 VJ=100.00
COMM 'EndPath S4614
COMM 'Path S4615
COMM SFTOF3D
COMM MOVJ C00158 BC00158 VJ=100.00  +MOVJ EC00158 VJ=100.00
COMM MOVL C00159 BC00159 V=800.0  +MOVJ EC00159 VJ=100.00
COMM SMOVL C00160 BC00160 V=166.7  +MOVJ EC00160
COMM SREFP 3 C00161 BC00161  +REFP EC00161
COMM CALL JOB:SEARCH-R1-S13D
COMM SET P034 P006
COMM SFTON3D P034
COMM SMOVL C00162 BC00162 V=166.7  +MOVJ EC00162
COMM SREFP 3 C00163 BC00163  +REFP EC00163
COMM CALL JOB:SEARCH-R1-S13D
COMM SET P034 P006
COMM SFTON3D P034
COMM SMOVL C00164 BC00164 V=166.7  +MOVJ EC00164
COMM SMOVL C00165 BC00165 V=166.7  +MOVJ EC00165
COMM SREFP 3 C00166 BC00166  +REFP EC00166
COMM CALL JOB:SEARCH-R1-S13D
COMM SET P034 P006
COMM SFTON3D P034
COMM SMOVL C00167 BC00167 V=166.7  +MOVJ EC00167
COMM MOVL C00168 BC00168 V=1000.0  +MOVJ EC00168 VJ=100.00
COMM 'EndPath S4615
COMM MOVJ C00169 BC00169 VJ=100.00  +MOVJ EC00169 VJ=100.00
COMM MOVJ C00170 BC00170 VJ=100.00  +MOVJ EC00170 VJ=100.00
COMM 'Path W4616
COMM SFTOF3D
COMM SFTON3D P026
COMM MOVJ C00171 BC00171 VJ=100.00  +MOVJ EC00171 VJ=100.00
COMM SMOVL C00172 BC00172 V=800.0  +MOVJ EC00172
COMM 'POPRAWIC!!!!
COMM SMOVL C00173 BC00173 V=166.7 PL=0  +MOVJ EC00173
COMM MACRO1 MJ#(0) ARGF21
COMM ARCON
COMM SWVON WEV#(100)
COMM SMOVL C00174 BC00174 V=9.2  +MOVJ EC00174
COMM SFTON3D P091
COMM SMOVL C00175 BC00175 V=9.2  +MOVJ EC00175
COMM SMOVL C00176 BC00176 V=9.2  +MOVJ EC00176
COMM SWVOF
COMM ARCOF
COMM SMOVL C00177 BC00177 V=800.0  +MOVJ EC00177
COMM SMOVL C00178 BC00178 V=1000.0  +MOVJ EC00178
COMM SFTOF3D
COMM 'EndPath W4616
COMM MOVJ C00179 BC00179 VJ=100.00  +MOVJ EC00179 VJ=100.00
COMM 'Path W4617
COMM SFTOF3D
COMM SFTON3D P028
COMM MOVJ C00180 BC00180 VJ=100.00  +MOVJ EC00180 VJ=100.00
COMM MOVJ C00181 BC00181 VJ=100.00  +MOVJ EC00181 VJ=100.00
COMM SMOVL C00182 BC00182 V=800.0  +MOVJ EC00182
COMM SMOVL C00183 BC00183 V=150.0 PL=0  +MOVJ EC00183
COMM ARCON
COMM SWVON WEV#(100)
COMM MOVL C00184 BC00184 V=9.2  +MOVJ EC00184 VJ=100.00
COMM SFTON3D P027
COMM SMOVL C00185 BC00185 V=9.2  +MOVJ EC00185
COMM SMOVL C00186 BC00186 V=9.2  +MOVJ EC00186
COMM ARCOF
COMM SWVOF
COMM SMOVL C00187 BC00187 V=800.0  +MOVJ EC00187
COMM SMOVL C00188 BC00188 V=1000.0  +MOVJ EC00188
COMM SFTOF3D
COMM 'EndPath W4617
COMM MOVJ C00189 BC00189 VJ=100.00  +MOVJ EC00189 VJ=100.00
COMM 'Path W4618
COMM SFTOF3D
COMM SFTON3D P022
COMM MOVJ C00190 BC00190 VJ=100.00  +MOVJ EC00190 VJ=100.00
COMM SMOVL C00191 BC00191 V=800.0  +MOVJ EC00191
COMM SMOVL C00192 BC00192 V=150.0 PL=0  +MOVJ EC00192
COMM MACRO1 MJ#(0) ARGF9
COMM ARCON
COMM SWVON WEV#(60)
COMM SFTON3D P021
COMM SMOVL C00193 BC00193 V=10.0  +MOVJ EC00193
COMM ARCOF
COMM SWVOF
COMM SMOVL C00194 BC00194 V=800.0  +MOVJ EC00194
COMM SMOVL C00195 BC00195 V=1000.0  +MOVJ EC00195
COMM SFTOF3D
COMM 'EndPath W4618
COMM 'Path W4883
COMM SFTOF3D
COMM SFTON3D P060
COMM MOVJ C00196 BC00196 VJ=100.00  +MOVJ EC00196 VJ=100.00
COMM SMOVL C00197 BC00197 V=800.0  +MOVJ EC00197
COMM SMOVL C00198 BC00198 V=150.0 PL=0  +MOVJ EC00198
COMM ARCON
COMM SMOVL C00199 BC00199 V=10.0  +MOVJ EC00199
COMM SMOVL C00200 BC00200 V=10.0  +MOVJ EC00200
COMM SMOVL C00201 BC00201 V=10.0  +MOVJ EC00201
COMM ARCOF
COMM SMOVL C00202 BC00202 V=800.0  +MOVJ EC00202
COMM SFTOF3D
COMM 'EndPath W4883
COMM 'Path W4884
COMM SFTOF3D
COMM SFTON3D P060
COMM SMOVL C00203 BC00203 V=800.0  +MOVJ EC00203
COMM SMOVL C00204 BC00204 V=150.0 PL=0  +MOVJ EC00204
COMM ARCON
COMM SMOVL C00205 BC00205 V=10.0  +MOVJ EC00205
COMM SMOVL C00206 BC00206 V=10.0  +MOVJ EC00206
COMM SMOVL C00207 BC00207 V=10.0  +MOVJ EC00207
COMM ARCOF
COMM SMOVL C00208 BC00208 V=800.0  +MOVJ EC00208
COMM SMOVL C00209 BC00209 V=1000.0  +MOVJ EC00209
COMM SFTOF3D
COMM 'EndPath W4884
COMM MOVJ C00210 BC00210 VJ=100.00  +MOVJ EC00210 VJ=100.00
COMM 'Path W4619
COMM SFTOF3D
COMM SFTON3D P030
COMM MOVJ C00211 BC00211 VJ=100.00  +MOVJ EC00211 VJ=100.00
COMM MOVJ C00212 BC00212 VJ=100.00  +MOVJ EC00212 VJ=100.00
COMM SMOVL C00213 BC00213 V=800.0  +MOVJ EC00213
COMM SMOVL C00214 BC00214 V=150.0 PL=0  +MOVJ EC00214
COMM ARCON
COMM MOVL C00215 BC00215 V=10.0  +MOVJ EC00215 VJ=100.00
COMM SFTON3D P029
COMM SMOVL C00216 BC00216 V=10.0  +MOVJ EC00216
COMM SMOVL C00217 BC00217 V=10.0  +MOVJ EC00217
COMM ARCOF
COMM SMOVL C00218 BC00218 V=800.0  +MOVJ EC00218
COMM SMOVL C00219 BC00219 V=1000.0  +MOVJ EC00219
COMM SFTOF3D
COMM 'EndPath W4619
COMM MOVJ C00220 BC00220 VJ=100.00  +MOVJ EC00220 VJ=100.00
COMM MOVJ C00221 BC00221 VJ=100.00  +MOVJ EC00221 VJ=100.00
COMM 'Path W4620
COMM SFTOF3D
COMM SFTON3D P033
COMM MOVJ C00222 BC00222 VJ=100.00  +MOVJ EC00222 VJ=100.00
COMM SMOVL C00223 BC00223 V=800.0  +MOVJ EC00223
COMM SMOVL C00224 BC00224 V=166.7 PL=0  +MOVJ EC00224
COMM ARCON
COMM SMOVL C00225 BC00225 V=9.2  +MOVJ EC00225
COMM SFTON3D P034
COMM SMOVL C00226 BC00226 V=9.2  +MOVJ EC00226
COMM SMOVL C00227 BC00227 V=9.2  +MOVJ EC00227
COMM ARCOF
COMM SMOVL C00228 BC00228 V=800.0  +MOVJ EC00228
COMM SMOVL C00229 BC00229 V=1000.0  +MOVJ EC00229
COMM SFTOF3D
COMM 'EndPath W4620
COMM MOVJ C00230 BC00230 VJ=100.00  +MOVJ EC00230 VJ=100.00
COMM 'Path W4621
COMM SFTOF3D
COMM SFTON3D P024
COMM MOVJ C00231 BC00231 VJ=100.00  +MOVJ EC00231 VJ=100.00
COMM SMOVL C00232 BC00232 V=800.0  +MOVJ EC00232
COMM SMOVL C00233 BC00233 V=166.7 PL=0  +MOVJ EC00233
COMM ARCON
COMM SMOVL C00234 BC00234 V=10.0  +MOVJ EC00234
COMM SFTON3D P025
COMM SMOVL C00235 BC00235 V=10.0  +MOVJ EC00235
COMM SMOVL C00236 BC00236 V=10.0  +MOVJ EC00236
COMM ARCOF
COMM SMOVL C00237 BC00237 V=800.0  +MOVJ EC00237
COMM SMOVL C00238 BC00238 V=1000.0  +MOVJ EC00238
COMM SFTOF3D
COMM 'EndPath W4621
COMM MOVJ C00239 BC00239 VJ=100.00  +MOVJ EC00239 VJ=100.00
COMM MOVJ C00240 BC00240 VJ=100.00  +MOVJ EC00240 VJ=100.00
COMM 'Path W4622
COMM SFTOF3D
COMM SFTON3D P032
COMM MOVJ C00241 BC00241 VJ=100.00  +MOVJ EC00241 VJ=100.00
COMM SMOVL C00242 BC00242 V=800.0  +MOVJ EC00242
COMM SMOVL C00243 BC00243 V=166.7 PL=0  +MOVJ EC00243
COMM ARCON
COMM SMOVL C00244 BC00244 V=9.2  +MOVJ EC00244
COMM SFTON3D P031
COMM SMOVL C00245 BC00245 V=9.2  +MOVJ EC00245
COMM SMOVL C00246 BC00246 V=9.2  +MOVJ EC00246
COMM ARCOF
COMM SMOVL C00247 BC00247 V=800.0  +MOVJ EC00247
COMM SMOVL C00248 BC00248 V=1000.0  +MOVJ EC00248
COMM SFTOF3D
COMM 'EndPath W4622
COMM 'Path W4623
COMM SFTOF3D
COMM SFTON3D P023
COMM MOVJ C00249 BC00249 VJ=100.00  +MOVJ EC00249 VJ=100.00
COMM JUMP *VVP
COMM MOVJ C00250 BC00250 VJ=100.00  +MOVJ EC00250 VJ=100.00
COMM SMOVL C00251 BC00251 V=800.0  +MOVJ EC00251
COMM SMOVL C00252 BC00252 V=166.7 PL=0  +MOVJ EC00252
COMM 'ARCON DO SPRAWDZENIA
COMM PAUSE
COMM SMOVL C00253 BC00253 V=10.0  +MOVJ EC00253
COMM SMOVL C00254 BC00254 V=10.0  +MOVJ EC00254
COMM SMOVL C00255 BC00255 V=10.0  +MOVJ EC00255
COMM SMOVL C00256 BC00256 V=10.0  +MOVJ EC00256
COMM SMOVL C00257 BC00257 V=10.0  +MOVJ EC00257
COMM SMOVL C00258 BC00258 V=10.0  +MOVJ EC00258
COMM SMOVL C00259 BC00259 V=10.0  +MOVJ EC00259
COMM SMOVL C00260 BC00260 V=10.0  +MOVJ EC00260
COMM SMOVL C00261 BC00261 V=10.0  +MOVJ EC00261
COMM ARCOF
COMM SMOVL C00262 BC00262 V=800.0  +MOVJ EC00262
COMM SMOVL C00263 BC00263 V=1000.0  +MOVJ EC00263
COMM SFTOF3D
COMM 'EndPath W4623
COMM 'Path W4624
COMM *VVP
COMM MOVJ C00264 BC00264 VJ=100.00  +MOVJ EC00264 VJ=100.00
COMM SFTOF3D
COMM SFTON3D P023
COMM MOVJ C00265 BC00265 VJ=100.00  +MOVJ EC00265 VJ=100.00
COMM SMOVL C00266 BC00266 V=800.0  +MOVJ EC00266
COMM SMOVL C00267 BC00267 V=150.0 PL=0  +MOVJ EC00267
COMM ARCON
COMM SMOVL C00268 BC00268 V=8.3  +MOVJ EC00268
COMM SMOVL C00269 BC00269 V=8.3  +MOVJ EC00269
COMM SMOVL C00270 BC00270 V=8.3  +MOVJ EC00270
COMM SMOVL C00271 BC00271 V=8.3  +MOVJ EC00271
COMM SMOVL C00272 BC00272 V=8.3  +MOVJ EC00272
COMM SMOVL C00273 BC00273 V=8.3  +MOVJ EC00273
COMM MOVL C00274 BC00274 V=8.3  +MOVJ EC00274 VJ=100.00
COMM ARCOF
COMM SMOVL C00275 BC00275 V=800.0  +MOVJ EC00275
COMM SMOVL C00276 BC00276 V=1000.0  +MOVJ EC00276
COMM SFTOF3D
COMM 'EndPath W4624
COMM MOVJ C00277 BC00277 VJ=100.00  +MOVJ EC00277 VJ=100.00
COMM 'Path S4625
COMM SFTOF3D
COMM CALL JOB:CLEAN-R1_KM_NEW
'X2_38-47,64(2)(90,0)
'Down
MOVJ C00278 BC00278 VJ=100.00  +MOVJ EC00278 VJ=100.00
'Up
'Path S4602
SFTOF3D
COMM MOVJ C00279 BC00279 VJ=100.00  +MOVJ EC00279 VJ=100.00
COMM MOVL C00280 BC00280 V=800.0  +MOVJ EC00280 VJ=100.00
COMM SMOVL C00281 BC00281 V=166.7  +MOVJ EC00281
COMM SREFP 3 C00282 BC00282  +REFP EC00282
COMM CALL JOB:SEARCH-R1-S13D
COMM SET P021 P006
COMM SFTON3D P021
COMM SMOVL C00283 BC00283 V=166.7  +MOVJ EC00283
COMM SREFP 3 C00284 BC00284  +REFP EC00284
COMM CALL JOB:SEARCH-R1-S13D
COMM SET P021 P006
COMM SFTON3D P021
COMM SMOVL C00285 BC00285 V=166.7  +MOVJ EC00285
COMM MOVL C00286 BC00286 V=1000.0  +MOVJ EC00286 VJ=100.00
COMM 'EndPath S4602
COMM 'Path S4603
COMM SFTOF3D
COMM MOVJ C00287 BC00287 VJ=100.00  +MOVJ EC00287 VJ=100.00
COMM MOVL C00288 BC00288 V=800.0  +MOVJ EC00288 VJ=100.00
COMM SMOVL C00289 BC00289 V=166.7  +MOVJ EC00289
COMM SREFP 3 C00290 BC00290  +REFP EC00290
COMM CALL JOB:SEARCH-R1-S13D
COMM SET P022 P006
COMM SFTON3D P022
COMM SMOVL C00291 BC00291 V=166.7  +MOVJ EC00291
COMM SREFP 3 C00292 BC00292  +REFP EC00292
COMM CALL JOB:SEARCH-R1-S13D
COMM SET P022 P006
COMM SFTON3D P022
COMM SMOVL C00293 BC00293 V=166.7  +MOVJ EC00293
COMM MOVL C00294 BC00294 V=1000.0  +MOVJ EC00294 VJ=100.00
COMM 'EndPath S4603
COMM 'Path S4604
COMM SFTOF3D
MOVJ C00295 BC00295 VJ=100.00  +MOVJ EC00295 VJ=100.00
MOVJ C00296 BC00296 VJ=100.00  +MOVJ EC00296 VJ=100.00
MOVL C00297 BC00297 V=800.0  +MOVJ EC00297 VJ=100.00
SMOVL C00298 BC00298 V=166.7  +MOVJ EC00298
SREFP 3 C00299 BC00299  +REFP EC00299
CALL JOB:SEARCH-R1-S13D
SET P023 P006
SFTON3D P023
SMOVL C00300 BC00300 V=166.7  +MOVJ EC00300
SREFP 3 C00301 BC00301  +REFP EC00301
CALL JOB:SEARCH-R1-S13D
SET P023 P006
SFTON3D P023
SMOVL C00302 BC00302 V=166.7  +MOVJ EC00302
SMOVL C00303 BC00303 V=333.3  +MOVJ EC00303
SMOVL C00304 BC00304 V=333.3  +MOVJ EC00304
SREFP 3 C00305 BC00305  +REFP EC00305
CALL JOB:SEARCH-R1-S13D
SET P023 P006
SFTON3D P023
SMOVL C00306 BC00306 V=166.7  +MOVJ EC00306
MOVL C00307 BC00307 V=1000.0  +MOVJ EC00307 VJ=100.00
'EndPath S4604
'Path S4605
SFTOF3D
MOVJ C00308 BC00308 VJ=100.00  +MOVJ EC00308 VJ=100.00
MOVL C00309 BC00309 V=800.0  +MOVJ EC00309 VJ=100.00
SMOVL C00310 BC00310 V=166.7  +MOVJ EC00310
SREFP 3 C00311 BC00311  +REFP EC00311
CALL JOB:SEARCH-R1-S13D
SET P024 P006
SFTON3D P024
SMOVL C00312 BC00312 V=166.7  +MOVJ EC00312
SMOVL C00313 BC00313 V=166.7  +MOVJ EC00313
SREFP 3 C00314 BC00314  +REFP EC00314
CALL JOB:SEARCH-R1-S13D
SET P024 P006
SFTON3D P024
SMOVL C00315 BC00315 V=166.7  +MOVJ EC00315
SMOVL C00316 BC00316 V=166.7  +MOVJ EC00316
SREFP 3 C00317 BC00317  +REFP EC00317
CALL JOB:SEARCH-R1-S13D
SET P024 P006
SFTON3D P024
SMOVL C00318 BC00318 V=166.7  +MOVJ EC00318
MOVL C00319 BC00319 V=1000.0  +MOVJ EC00319 VJ=100.00
MOVL C00320 BC00320 V=1000.0  +MOVJ EC00320 VJ=100.00
'EndPath S4605
'Path S4606
SFTOF3D
MOVJ C00321 BC00321 VJ=100.00  +MOVJ EC00321 VJ=100.00
MOVL C00322 BC00322 V=800.0  +MOVJ EC00322 VJ=100.00
SMOVL C00323 BC00323 V=166.7  +MOVJ EC00323
SREFP 3 C00324 BC00324  +REFP EC00324
CALL JOB:SEARCH-R1-S13D
SET P025 P006
SFTON3D P025
SMOVL C00325 BC00325 V=166.7  +MOVJ EC00325
SREFP 3 C00326 BC00326  +REFP EC00326
CALL JOB:SEARCH-R1-S13D
SET P025 P006
SFTON3D P025
SMOVL C00327 BC00327 V=166.7  +MOVJ EC00327
SMOVL C00328 BC00328 V=166.7  +MOVJ EC00328
SREFP 3 C00329 BC00329  +REFP EC00329
CALL JOB:SEARCH-R1-S13D
SET P025 P006
SFTON3D P025
SMOVL C00330 BC00330 V=166.7  +MOVJ EC00330
MOVL C00331 BC00331 V=1000.0  +MOVJ EC00331 VJ=100.00
MOVL C00332 BC00332 V=1000.0  +MOVJ EC00332 VJ=100.00
'EndPath S4606
'Path S4607
SFTOF3D
MOVJ C00333 BC00333 VJ=100.00  +MOVJ EC00333 VJ=100.00
MOVL C00334 BC00334 V=800.0  +MOVJ EC00334 VJ=100.00
SMOVL C00335 BC00335 V=166.7  +MOVJ EC00335
SREFP 3 C00336 BC00336  +REFP EC00336
CALL JOB:SEARCH-R1-S13D
SET P026 P006
SFTON3D P026
SMOVL C00337 BC00337 V=166.7  +MOVJ EC00337
SREFP 3 C00338 BC00338  +REFP EC00338
CALL JOB:SEARCH-R1-S13D
SET P026 P006
SFTON3D P026
SMOVL C00339 BC00339 V=166.7  +MOVJ EC00339
MOVL C00340 BC00340 V=1000.0  +MOVJ EC00340 VJ=100.00
SFTOF3D
SMOVL C00341 BC00341 V=166.7  +MOVJ EC00341
SREFP 3 C00342 BC00342  +REFP EC00342
CALL JOB:SEARCH-R1-S13D
SET P091 P006
SFTON3D P091
SMOVL C00343 BC00343 V=166.7  +MOVJ EC00343
SREFP 3 C00344 BC00344  +REFP EC00344
CALL JOB:SEARCH-R1-S13D
SET P091 P006
SFTON3D P091
SMOVL C00345 BC00345 V=166.7  +MOVJ EC00345
SMOVL C00346 BC00346 V=500.0  +MOVJ EC00346
'EndPath S4607
MOVJ C00347 BC00347 VJ=100.00  +MOVJ EC00347 VJ=100.00
MOVJ C00348 BC00348 VJ=100.00  +MOVJ EC00348 VJ=100.00
'Path S4608
SFTOF3D
MOVJ C00349 BC00349 VJ=100.00  +MOVJ EC00349 VJ=100.00
MOVL C00350 BC00350 V=800.0  +MOVJ EC00350 VJ=100.00
SMOVL C00351 BC00351 V=166.7  +MOVJ EC00351
SREFP 3 C00352 BC00352  +REFP EC00352
CALL JOB:SEARCH-R1-S13D
SET P027 P006
SFTON3D P027
SMOVL C00353 BC00353 V=166.7  +MOVJ EC00353
SMOVL C00354 BC00354 V=166.7  +MOVJ EC00354
SREFP 3 C00355 BC00355  +REFP EC00355
CALL JOB:SEARCH-R1-S13D
SET P027 P006
SFTON3D P027
SMOVL C00356 BC00356 V=166.7  +MOVJ EC00356
SMOVL C00357 BC00357 V=166.7  +MOVJ EC00357
SREFP 3 C00358 BC00358  +REFP EC00358
CALL JOB:SEARCH-R1-S13D
SET P027 P006
SFTON3D P027
SMOVL C00359 BC00359 V=166.7  +MOVJ EC00359
MOVL C00360 BC00360 V=1000.0  +MOVJ EC00360 VJ=100.00
MOVL C00361 BC00361 V=1000.0  +MOVJ EC00361 VJ=100.00
'EndPath S4608
'Path S4609
SFTOF3D
MOVJ C00362 BC00362 VJ=100.00  +MOVJ EC00362 VJ=100.00
MOVL C00363 BC00363 V=800.0  +MOVJ EC00363 VJ=100.00
